LIN {X 0,Y 368.937,Z 294.527,A -85,B 0,C 180,E1 -12892.391,E2 -12892.391} C_VEL
LIN {X 0,Y 368.985,Z 294.519,A -85,B 0,C 180,E1 -12895.977,E2 -12895.977} C_VEL
LIN {X 0,Y 368.95,Z 294.527,A -85,B 0,C 180,E1 -12898.81,E2 -12898.81} C_VEL
LIN {X 0,Y 368.88,Z 294.532,A -85,B 0,C 180,E1 -12902.234,E2 -12902.234} C_VEL
LIN {X 0,Y 368.907,Z 294.534,A -85,B 0,C 180,E1 -12904.998,E2 -12904.998} C_VEL
LIN {X 0,Y 368.889,Z 294.533,A -85,B 0,C 180,E1 -12908.637,E2 -12908.637} C_VEL
LIN {X 0,Y 368.962,Z 294.67,A -85,B 0,C 180,E1 -12910.272,E2 -12910.272} C_VEL
LIN {X 0,Y 369.512,Z 297.416,A -85,B 0,C 180,E1 -12911.001,E2 -12911.001} C_VEL
LIN {X 0,Y 374.72,Z 313.747,A -85,B 0,C 180,E1 -12911.64,E2 -12911.64} C_VEL
LIN {X 0,Y 375.92,Z 320.785,A -85,B 0,C 180,E1 -12911.859,E2 -12911.859} C_VEL
LIN {X 0,Y 375.904,Z 322.653,A -85,B 0,C 180,E1 -12911.902,E2 -12911.902} C_VEL
LIN {X 0,Y 375.086,Z 328.475,A -85,B 0,C 180,E1 -12911.998,E2 -12911.998} C_VEL
LIN {X 0,Y 369.16,Z 347.372,A -85,B 0,C 180,E1 -12912.166,E2 -12912.166} C_VEL
LIN {X 0,Y 368.425,Z 353.191,A -85,B 0,C 180,E1 -12912.271,E2 -12912.271} C_VEL
LIN {X 0,Y 367.241,Z 406.595,A -85,B 0,C 180,E1 -12913.49,E2 -12913.49} C_VEL
LIN {X 0,Y 366.848,Z 418.98,A -85,B 0,C 180,E1 -12913.978,E2 -12913.978} C_VEL
LIN {X 0,Y 366.221,Z 431.276,A -85,B 0,C 180,E1 -12914.664,E2 -12914.664} C_VEL
LIN {X 0,Y 365.574,Z 442.837,A -85,B 0,C 180,E1 -12915.53,E2 -12915.53} C_VEL
LIN {X 0,Y 364.747,Z 453.885,A -85,B 0,C 180,E1 -12916.579,E2 -12916.579} C_VEL
LIN {X 0,Y 363.922,Z 464.624,A -85,B 0,C 180,E1 -12917.85,E2 -12917.85} C_VEL
LIN {X 0,Y 363.098,Z 474.262,A -85,B 0,C 180,E1 -12919.27,E2 -12919.27} C_VEL
LIN {X 0,Y 362.367,Z 483.022,A -85,B 0,C 180,E1 -12920.867,E2 -12920.867} C_VEL
LIN {X 0,Y 361.726,Z 490.562,A -85,B 0,C 180,E1 -12922.57,E2 -12922.57} C_VEL
LIN {X 0,Y 361.27,Z 496.591,A -85,B 0,C 180,E1 -12924.296,E2 -12924.296} C_VEL
LIN {X 0,Y 360.869,Z 501.916,A -85,B 0,C 180,E1 -12926.288,E2 -12926.288} C_VEL
LIN {X 0,Y 360.532,Z 505.675,A -85,B 0,C 180,E1 -12928.243,E2 -12928.243} C_VEL
LIN {X 0,Y 360.404,Z 507.362,A -85,B 0,C 180,E1 -12929.536,E2 -12929.536} C_VEL
LIN {X 0,Y 360.357,Z 508.805,A -85,B 0,C 180,E1 -12931.343,E2 -12931.343} C_VEL
LIN {X 0,Y 360.365,Z 509.152,A -85,B 0,C 180,E1 -12933.35,E2 -12933.35} C_VEL
LIN {X 0,Y 360.486,Z 508.683,A -85,B 0,C 180,E1 -12934.602,E2 -12934.602} C_VEL
LIN {X 0,Y 360.749,Z 507.241,A -85,B 0,C 180,E1 -12936.279,E2 -12936.279} C_VEL
LIN {X 0,Y 361.198,Z 504.193,A -85,B 0,C 180,E1 -12938.304,E2 -12938.304} C_VEL
LIN {X 0,Y 361.664,Z 500.21,A -85,B 0,C 180,E1 -12940.12,E2 -12940.12} C_VEL
LIN {X 0,Y 362.37,Z 494.924,A -85,B 0,C 180,E1 -12941.923,E2 -12941.923} C_VEL
LIN {X 0,Y 363.289,Z 488.133,A -85,B 0,C 180,E1 -12943.71,E2 -12943.71} C_VEL
LIN {X 0,Y 364.388,Z 479.592,A -85,B 0,C 180,E1 -12945.48,E2 -12945.48} C_VEL
LIN {X 0,Y 365.473,Z 470.795,A -85,B 0,C 180,E1 -12946.942,E2 -12946.942} C_VEL
LIN {X 0,Y 366.712,Z 460.323,A -85,B 0,C 180,E1 -12948.331,E2 -12948.331} C_VEL
LIN {X 0,Y 367.803,Z 449.016,A -85,B 0,C 180,E1 -12949.542,E2 -12949.542} C_VEL
LIN {X 0,Y 368.872,Z 436.91,A -85,B 0,C 180,E1 -12950.542,E2 -12950.542} C_VEL
LIN {X 0,Y 369.659,Z 424.92,A -85,B 0,C 180,E1 -12951.302,E2 -12951.302} C_VEL
LIN {X 0,Y 370.291,Z 412.735,A -85,B 0,C 180,E1 -12951.86,E2 -12951.86} C_VEL
LIN {X 0,Y 370.758,Z 397.567,A -85,B 0,C 180,E1 -12952.291,E2 -12952.291} C_VEL
LIN {X 0,Y 373.067,Z 321.948,A -85,B 0,C 180,E1 -12954.082,E2 -12954.082} C_VEL
LIN {X 0,Y 367.77,Z 308.846,A -85,B 0,C 180,E1 -12954.896,E2 -12954.896} C_VEL
LIN {X 0,Y 362.98,Z 299.287,A -85,B 0,C 180,E1 -12955.628,E2 -12955.628} C_VEL
LIN {X 0,Y 362.025,Z 295.396,A -85,B 0,C 180,E1 -12956.592,E2 -12956.592} C_VEL
LIN {X 0,Y 362.232,Z 295.369,A -85,B 0,C 180,E1 -12957.777,E2 -12957.777} C_VEL
LIN {X 0,Y 362.377,Z 295.346,A -85,B 0,C 180,E1 -12960.001,E2 -12960.001} C_VEL
LIN {X 0,Y 362.232,Z 295.365,A -85,B 0,C 180,E1 -12962.224,E2 -12962.224} C_VEL
LIN {X 0,Y 362.112,Z 295.379,A -85,B 0,C 180,E1 -12966.688,E2 -12966.688} C_VEL
LIN {X 0,Y 361.986,Z 295.393,A -85,B 0,C 180,E1 -12970.064,E2 -12970.064} C_VEL
LIN {X 0,Y 361.953,Z 295.398,A -85,B 0,C 180,E1 -12973.9,E2 -12973.9} C_VEL
LIN {X 0,Y 361.883,Z 295.406,A -85,B 0,C 180,E1 -12976.937,E2 -12976.937} C_VEL
LIN {X 0,Y 361.832,Z 295.407,A -85,B 0,C 180,E1 -12980.465,E2 -12980.465} C_VEL
LIN {X 0,Y 361.854,Z 295.409,A -85,B 0,C 180,E1 -12984.116,E2 -12984.116} C_VEL
LIN {X 0,Y 361.901,Z 295.401,A -85,B 0,C 180,E1 -12986.724,E2 -12986.724} C_VEL
LIN {X 0,Y 361.815,Z 295.415,A -85,B 0,C 180,E1 -12990.334,E2 -12990.334} C_VEL
LIN {X 0,Y 361.82,Z 295.41,A -85,B 0,C 180,E1 -12994.285,E2 -12994.285} C_VEL
LIN {X 0,Y 361.833,Z 295.41,A -85,B 0,C 180,E1 -12997.227,E2 -12997.227} C_VEL
LIN {X 0,Y 361.841,Z 295.412,A -85,B 0,C 180,E1 -13000.766,E2 -13000.766} C_VEL
LIN {X 0,Y 361.79,Z 295.416,A -85,B 0,C 180,E1 -13004.373,E2 -13004.373} C_VEL
LIN {X 0,Y 361.812,Z 295.419,A -85,B 0,C 180,E1 -13007.573,E2 -13007.573} C_VEL
LIN {X 0,Y 361.845,Z 295.412,A -85,B 0,C 180,E1 -13010.979,E2 -13010.979} C_VEL
LIN {X 0,Y 361.857,Z 295.415,A -85,B 0,C 180,E1 -13014.66,E2 -13014.66} C_VEL
LIN {X 0,Y 361.893,Z 295.418,A -85,B 0,C 180,E1 -13018.3,E2 -13018.3} C_VEL
LIN {X 0,Y 364.588,Z 305.964,A -85,B 0,C 180,E1 -13020.915,E2 -13020.915} C_VEL
LIN {X 0,Y 366.627,Z 315.872,A -85,B 0,C 180,E1 -13023.23,E2 -13023.23} C_VEL
LIN {X 0,Y 366.76,Z 318.771,A -85,B 0,C 180,E1 -13023.854,E2 -13023.854} C_VEL
LIN {X 0,Y 365.434,Z 332.937,A -85,B 0,C 180,E1 -13026.691,E2 -13026.691} C_VEL
LIN {X 0,Y 369.47,Z 354.155,A -85,B 0,C 180,E1 -13027.61,E2 -13027.61} C_VEL
LIN {X 0,Y 371.571,Z 370.409,A -85,B 0,C 180,E1 -13028.205,E2 -13028.205} C_VEL
LIN {X 0,Y 371.845,Z 375.745,A -85,B 0,C 180,E1 -13028.366,E2 -13028.366} C_VEL
LIN {X 0,Y 369.813,Z 444.426,A -85,B 0,C 180,E1 -13030.001,E2 -13030.001} C_VEL
LIN {X 0,Y 368.911,Z 458.053,A -85,B 0,C 180,E1 -13030.529,E2 -13030.529} C_VEL
LIN {X 0,Y 367.912,Z 470.015,A -85,B 0,C 180,E1 -13031.199,E2 -13031.199} C_VEL
LIN {X 0,Y 366.675,Z 482.615,A -85,B 0,C 180,E1 -13032.145,E2 -13032.145} C_VEL
LIN {X 0,Y 365.448,Z 493.967,A -85,B 0,C 180,E1 -13033.237,E2 -13033.237} C_VEL
LIN {X 0,Y 364.248,Z 504.34,A -85,B 0,C 180,E1 -13034.483,E2 -13034.483} C_VEL
LIN {X 0,Y 363.079,Z 514.461,A -85,B 0,C 180,E1 -13036.001,E2 -13036.001} C_VEL
LIN {X 0,Y 362.119,Z 523.48,A -85,B 0,C 180,E1 -13037.676,E2 -13037.676} C_VEL
LIN {X 0,Y 361.285,Z 530.704,A -85,B 0,C 180,E1 -13039.353,E2 -13039.353} C_VEL
LIN {X 0,Y 360.817,Z 536.522,A -85,B 0,C 180,E1 -13041.038,E2 -13041.038} C_VEL
LIN {X 0,Y 360.565,Z 541.13,A -85,B 0,C 180,E1 -13042.724,E2 -13042.724} C_VEL
LIN {X 0,Y 360.397,Z 544.627,A -85,B 0,C 180,E1 -13044.407,E2 -13044.407} C_VEL
LIN {X 0,Y 360.407,Z 546.388,A -85,B 0,C 180,E1 -13045.529,E2 -13045.529} C_VEL
LIN {X 0,Y 360.364,Z 547.727,A -85,B 0,C 180,E1 -13046.648,E2 -13046.648} C_VEL
LIN {X 0,Y 360.43,Z 548.607,A -85,B 0,C 180,E1 -13047.767,E2 -13047.767} C_VEL
LIN {X 0,Y 360.52,Z 549.064,A -85,B 0,C 180,E1 -13048.885,E2 -13048.885} C_VEL
LIN {X 0,Y 360.523,Z 549.11,A -85,B 0,C 180,E1 -13050.002,E2 -13050.002} C_VEL
LIN {X 0,Y 360.533,Z 548.742,A -85,B 0,C 180,E1 -13051.119,E2 -13051.119} C_VEL
LIN {X 0,Y 360.503,Z 547.904,A -85,B 0,C 180,E1 -13052.236,E2 -13052.236} C_VEL
LIN {X 0,Y 360.398,Z 546.633,A -85,B 0,C 180,E1 -13053.355,E2 -13053.355} C_VEL
LIN {X 0,Y 360.479,Z 543.903,A -85,B 0,C 180,E1 -13055.034,E2 -13055.034} C_VEL
LIN {X 0,Y 360.57,Z 540.082,A -85,B 0,C 180,E1 -13056.717,E2 -13056.717} C_VEL
LIN {X 0,Y 360.697,Z 535.07,A -85,B 0,C 180,E1 -13058.404,E2 -13058.404} C_VEL
LIN {X 0,Y 361.053,Z 528.729,A -85,B 0,C 180,E1 -13060.09,E2 -13060.09} C_VEL
LIN {X 0,Y 361.659,Z 520.778,A -85,B 0,C 180,E1 -13061.774,E2 -13061.774} C_VEL
LIN {X 0,Y 362.295,Z 512.626,A -85,B 0,C 180,E1 -13063.176,E2 -13063.176} C_VEL
LIN {X 0,Y 363.086,Z 502.676,A -85,B 0,C 180,E1 -13064.574,E2 -13064.574} C_VEL
LIN {X 0,Y 364.013,Z 491.591,A -85,B 0,C 180,E1 -13065.826,E2 -13065.826} C_VEL
LIN {X 0,Y 365.001,Z 479.007,A -85,B 0,C 180,E1 -13066.932,E2 -13066.932} C_VEL
LIN {X 0,Y 365.887,Z 466.723,A -85,B 0,C 180,E1 -13067.754,E2 -13067.754} C_VEL
LIN {X 0,Y 366.652,Z 453.074,A -85,B 0,C 180,E1 -13068.401,E2 -13068.401} C_VEL
LIN {X 0,Y 367.187,Z 439.632,A -85,B 0,C 180,E1 -13068.807,E2 -13068.807} C_VEL
LIN {X 0,Y 368.409,Z 371.766,A -85,B 0,C 180,E1 -13070.329,E2 -13070.329} C_VEL
LIN {X 0,Y 363.954,Z 336.994,A -85,B 0,C 180,E1 -13071.386,E2 -13071.386} C_VEL
LIN {X 0,Y 365.627,Z 318.277,A -85,B 0,C 180,E1 -13075.387,E2 -13075.387} C_VEL
LIN {X 0,Y 365.717,Z 314.433,A -85,B 0,C 180,E1 -13076.23,E2 -13076.23} C_VEL
LIN {X 0,Y 363.066,Z 300.891,A -85,B 0,C 180,E1 -13079.414,E2 -13079.414} C_VEL
LIN {X 0,Y 361.884,Z 295.409,A -85,B 0,C 180,E1 -13080.783,E2 -13080.783} C_VEL
LIN {X 0,Y 361.846,Z 295.412,A -85,B 0,C 180,E1 -13084.279,E2 -13084.279} C_VEL
LIN {X 0,Y 361.851,Z 295.41,A -85,B 0,C 180,E1 -13087.219,E2 -13087.219} C_VEL
LIN {X 0,Y 361.803,Z 295.42,A -85,B 0,C 180,E1 -13090.749,E2 -13090.749} C_VEL
LIN {X 0,Y 361.8,Z 295.416,A -85,B 0,C 180,E1 -13094.368,E2 -13094.368} C_VEL
LIN {X 0,Y 361.81,Z 295.414,A -85,B 0,C 180,E1 -13097.569,E2 -13097.569} C_VEL
LIN {X 0,Y 361.827,Z 295.412,A -85,B 0,C 180,E1 -13101.57,E2 -13101.57} C_VEL
LIN {X 0,Y 361.854,Z 295.411,A -85,B 0,C 180,E1 -13104.655,E2 -13104.655} C_VEL
LIN {X 0,Y 361.829,Z 295.416,A -85,B 0,C 180,E1 -13107.053,E2 -13107.053} C_VEL
LIN {X 0,Y 361.849,Z 295.414,A -85,B 0,C 180,E1 -13110.95,E2 -13110.95} C_VEL
LIN {X 0,Y 361.863,Z 295.409,A -85,B 0,C 180,E1 -13114.705,E2 -13114.705} C_VEL
LIN {X 0,Y 361.832,Z 295.411,A -85,B 0,C 180,E1 -13118.343,E2 -13118.343} C_VEL
LIN {X 0,Y 361.897,Z 295.403,A -85,B 0,C 180,E1 -13122.084,E2 -13122.084} C_VEL
LIN {X 0,Y 361.937,Z 295.402,A -85,B 0,C 180,E1 -13125.378,E2 -13125.378} C_VEL
LIN {X 0,Y 361.945,Z 295.398,A -85,B 0,C 180,E1 -13128.803,E2 -13128.803} C_VEL
LIN {X 0,Y 362.09,Z 295.379,A -85,B 0,C 180,E1 -13132.191,E2 -13132.191} C_VEL
LIN {X 0,Y 362.083,Z 295.38,A -85,B 0,C 180,E1 -13134.43,E2 -13134.43} C_VEL
LIN {X 0,Y 362.249,Z 295.362,A -85,B 0,C 180,E1 -13137.776,E2 -13137.776} C_VEL
LIN {X 0,Y 362.356,Z 295.347,A -85,B 0,C 180,E1 -13139.999,E2 -13139.999} C_VEL
LIN {X 0,Y 362.249,Z 295.36,A -85,B 0,C 180,E1 -13142.223,E2 -13142.223} C_VEL
LIN {X 0,Y 362.129,Z 295.374,A -85,B 0,C 180,E1 -13146.686,E2 -13146.686} C_VEL
LIN {X 0,Y 362.006,Z 295.391,A -85,B 0,C 180,E1 -13150.062,E2 -13150.062} C_VEL
LIN {X 0,Y 361.973,Z 295.397,A -85,B 0,C 180,E1 -13153.898,E2 -13153.898} C_VEL
LIN {X 0,Y 361.901,Z 295.403,A -85,B 0,C 180,E1 -13156.935,E2 -13156.935} C_VEL
LIN {X 0,Y 361.851,Z 295.409,A -85,B 0,C 180,E1 -13160.462,E2 -13160.462} C_VEL
LIN {X 0,Y 361.872,Z 295.409,A -85,B 0,C 180,E1 -13164.114,E2 -13164.114} C_VEL
LIN {X 0,Y 361.92,Z 295.4,A -85,B 0,C 180,E1 -13166.722,E2 -13166.722} C_VEL
LIN {X 0,Y 361.855,Z 295.41,A -85,B 0,C 180,E1 -13170.329,E2 -13170.329} C_VEL
LIN {X 0,Y 361.835,Z 295.414,A -85,B 0,C 180,E1 -13174.282,E2 -13174.282} C_VEL
LIN {X 0,Y 361.847,Z 295.41,A -85,B 0,C 180,E1 -13177.224,E2 -13177.224} C_VEL
LIN {X 0,Y 361.853,Z 295.409,A -85,B 0,C 180,E1 -13180.762,E2 -13180.762} C_VEL
LIN {X 0,Y 361.829,Z 295.415,A -85,B 0,C 180,E1 -13184.366,E2 -13184.366} C_VEL
LIN {X 0,Y 361.871,Z 295.408,A -85,B 0,C 180,E1 -13187.561,E2 -13187.561} C_VEL
LIN {X 0,Y 361.863,Z 295.408,A -85,B 0,C 180,E1 -13190.974,E2 -13190.974} C_VEL
LIN {X 0,Y 361.865,Z 295.409,A -85,B 0,C 180,E1 -13194.656,E2 -13194.656} C_VEL
LIN {X 0,Y 361.83,Z 295.416,A -85,B 0,C 180,E1 -13198.371,E2 -13198.371} C_VEL
LIN {X 0,Y 361.902,Z 295.406,A -85,B 0,C 180,E1 -13202.221,E2 -13202.221} C_VEL
LIN {X 0,Y 361.923,Z 295.402,A -85,B 0,C 180,E1 -13204.71,E2 -13204.71} C_VEL
LIN {X 0,Y 361.888,Z 295.408,A -85,B 0,C 180,E1 -13208.347,E2 -13208.347} C_VEL
LIN {X 0,Y 361.964,Z 295.398,A -85,B 0,C 180,E1 -13212.061,E2 -13212.061} C_VEL
LIN {X 0,Y 361.995,Z 295.394,A -85,B 0,C 180,E1 -13216.101,E2 -13216.101} C_VEL
LIN {X 0,Y 362.029,Z 295.388,A -85,B 0,C 180,E1 -13219.937,E2 -13219.937} C_VEL
LIN {X 0,Y 362.149,Z 295.374,A -85,B 0,C 180,E1 -13222.192,E2 -13222.192} C_VEL
LIN {X 0,Y 362.116,Z 295.379,A -85,B 0,C 180,E1 -13224.43,E2 -13224.43} C_VEL
LIN {X 0,Y 362.28,Z 295.355,A -85,B 0,C 180,E1 -13227.775,E2 -13227.775} C_VEL
LIN {X 0,Y 362.425,Z 295.338,A -85,B 0,C 180,E1 -13229.998,E2 -13229.998} C_VEL
LIN {X 0,Y 362.28,Z 295.357,A -85,B 0,C 180,E1 -13232.222,E2 -13232.222} C_VEL
LIN {X 0,Y 362.165,Z 295.374,A -85,B 0,C 180,E1 -13236.684,E2 -13236.684} C_VEL
LIN {X 0,Y 362.069,Z 295.386,A -85,B 0,C 180,E1 -13238.931,E2 -13238.931} C_VEL
LIN {X 0,Y 361.959,Z 295.397,A -85,B 0,C 180,E1 -13242.329,E2 -13242.329} C_VEL
LIN {X 0,Y 361.954,Z 295.399,A -85,B 0,C 180,E1 -13244.617,E2 -13244.617} C_VEL
LIN {X 0,Y 361.951,Z 295.396,A -85,B 0,C 180,E1 -13248.096,E2 -13248.096} C_VEL
LIN {X 0,Y 361.902,Z 295.402,A -85,B 0,C 180,E1 -13251.648,E2 -13251.648} C_VEL
LIN {X 0,Y 361.914,Z 295.403,A -85,B 0,C 180,E1 -13255.286,E2 -13255.286} C_VEL
LIN {X 0,Y 361.906,Z 295.401,A -85,B 0,C 180,E1 -13257.774,E2 -13257.774} C_VEL
LIN {X 0,Y 361.828,Z 295.415,A -85,B 0,C 180,E1 -13261.282,E2 -13261.282} C_VEL
LIN {X 0,Y 361.833,Z 295.41,A -85,B 0,C 180,E1 -13264.277,E2 -13264.277} C_VEL
LIN {X 0,Y 361.848,Z 295.414,A -85,B 0,C 180,E1 -13267.221,E2 -13267.221} C_VEL
LIN {X 0,Y 361.916,Z 295.43,A -85,B 0,C 180,E1 -13270.017,E2 -13270.017} C_VEL
LIN {X 0,Y 362.382,Z 297.887,A -85,B 0,C 180,E1 -13270.663,E2 -13270.663} C_VEL
LIN {X 0,Y 368.104,Z 315.692,A -85,B 0,C 180,E1 -13271.374,E2 -13271.374} C_VEL
LIN {X 0,Y 369.116,Z 321.233,A -85,B 0,C 180,E1 -13271.554,E2 -13271.554} C_VEL
LIN {X 0,Y 368.425,Z 353.191,A -85,B 0,C 180,E1 -13272.271,E2 -13272.271} C_VEL
LIN {X 0,Y 367.673,Z 359.015,A -85,B 0,C 180,E1 -13272.374,E2 -13272.374} C_VEL
LIN {X 0,Y 361.662,Z 377.908,A -85,B 0,C 180,E1 -13272.548,E2 -13272.548} C_VEL
LIN {X 0,Y 360.879,Z 383.734,A -85,B 0,C 180,E1 -13272.652,E2 -13272.652} C_VEL
LIN {X 0,Y 360.342,Z 407.807,A -85,B 0,C 180,E1 -13273.244,E2 -13273.244} C_VEL
LIN {X 0,Y 359.954,Z 420.001,A -85,B 0,C 180,E1 -13273.747,E2 -13273.747} C_VEL
LIN {X 0,Y 359.306,Z 432.235,A -85,B 0,C 180,E1 -13274.454,E2 -13274.454} C_VEL
LIN {X 0,Y 358.622,Z 443.582,A -85,B 0,C 180,E1 -13275.329,E2 -13275.329} C_VEL
LIN {X 0,Y 357.785,Z 454.352,A -85,B 0,C 180,E1 -13276.374,E2 -13276.374} C_VEL
LIN {X 0,Y 356.973,Z 464.554,A -85,B 0,C 180,E1 -13277.601,E2 -13277.601} C_VEL
LIN {X 0,Y 356.132,Z 474.289,A -85,B 0,C 180,E1 -13279.045,E2 -13279.045} C_VEL
LIN {X 0,Y 355.332,Z 483.423,A -85,B 0,C 180,E1 -13280.735,E2 -13280.735} C_VEL
LIN {X 0,Y 354.687,Z 490.753,A -85,B 0,C 180,E1 -13282.417,E2 -13282.417} C_VEL
LIN {X 0,Y 354.243,Z 496.343,A -85,B 0,C 180,E1 -13284.014,E2 -13284.014} C_VEL
LIN {X 0,Y 353.898,Z 500.604,A -85,B 0,C 180,E1 -13285.531,E2 -13285.531} C_VEL
LIN {X 0,Y 353.769,Z 502.956,A -85,B 0,C 180,E1 -13286.539,E2 -13286.539} C_VEL
LIN {X 0,Y 353.567,Z 504.904,A -85,B 0,C 180,E1 -13287.542,E2 -13287.542} C_VEL
LIN {X 0,Y 353.376,Z 506.929,A -85,B 0,C 180,E1 -13288.863,E2 -13288.863} C_VEL
LIN {X 0,Y 353.28,Z 509.047,A -85,B 0,C 180,E1 -13291.068,E2 -13291.068} C_VEL
LIN {X 0,Y 353.275,Z 509.616,A -85,B 0,C 180,E1 -13292.771,E2 -13292.771} C_VEL
LIN {X 0,Y 353.357,Z 509.404,A -85,B 0,C 180,E1 -13294.052,E2 -13294.052} C_VEL
LIN {X 0,Y 353.625,Z 508.047,A -85,B 0,C 180,E1 -13296.076,E2 -13296.076} C_VEL
LIN {X 0,Y 354.027,Z 505.768,A -85,B 0,C 180,E1 -13297.842,E2 -13297.842} C_VEL
LIN {X 0,Y 354.491,Z 502.228,A -85,B 0,C 180,E1 -13299.7,E2 -13299.7} C_VEL
LIN {X 0,Y 355.227,Z 496.869,A -85,B 0,C 180,E1 -13301.719,E2 -13301.719} C_VEL
LIN {X 0,Y 356.237,Z 489.977,A -85,B 0,C 180,E1 -13303.673,E2 -13303.673} C_VEL
LIN {X 0,Y 357.363,Z 481.801,A -85,B 0,C 180,E1 -13305.479,E2 -13305.479} C_VEL
LIN {X 0,Y 358.469,Z 473.4,A -85,B 0,C 180,E1 -13306.97,E2 -13306.97} C_VEL
LIN {X 0,Y 359.681,Z 463.925,A -85,B 0,C 180,E1 -13308.339,E2 -13308.339} C_VEL
LIN {X 0,Y 360.948,Z 452.806,A -85,B 0,C 180,E1 -13309.625,E2 -13309.625} C_VEL
LIN {X 0,Y 361.948,Z 441.756,A -85,B 0,C 180,E1 -13310.642,E2 -13310.642} C_VEL
LIN {X 0,Y 362.973,Z 429.197,A -85,B 0,C 180,E1 -13311.532,E2 -13311.532} C_VEL
LIN {X 0,Y 363.688,Z 416.105,A -85,B 0,C 180,E1 -13312.201,E2 -13312.201} C_VEL
LIN {X 0,Y 364.188,Z 403.673,A -85,B 0,C 180,E1 -13312.621,E2 -13312.621} C_VEL
LIN {X 0,Y 366.868,Z 323.745,A -85,B 0,C 180,E1 -13314.561,E2 -13314.561} C_VEL
LIN {X 0,Y 361.403,Z 310.693,A -85,B 0,C 180,E1 -13315.422,E2 -13315.422} C_VEL
LIN {X 0,Y 355.957,Z 299.947,A -85,B 0,C 180,E1 -13316.286,E2 -13316.286} C_VEL
LIN {X 0,Y 355.09,Z 296.259,A -85,B 0,C 180,E1 -13317.235,E2 -13317.235} C_VEL
LIN {X 0,Y 355.326,Z 296.224,A -85,B 0,C 180,E1 -13320.001,E2 -13320.001} C_VEL
LIN {X 0,Y 355.196,Z 296.242,A -85,B 0,C 180,E1 -13322.268,E2 -13322.268} C_VEL
LIN {X 0,Y 355.076,Z 296.256,A -85,B 0,C 180,E1 -13326.821,E2 -13326.821} C_VEL
LIN {X 0,Y 354.933,Z 296.271,A -85,B 0,C 180,E1 -13330.266,E2 -13330.266} C_VEL
LIN {X 0,Y 354.898,Z 296.277,A -85,B 0,C 180,E1 -13334.02,E2 -13334.02} C_VEL
LIN {X 0,Y 354.846,Z 296.279,A -85,B 0,C 180,E1 -13338.094,E2 -13338.094} C_VEL
LIN {X 0,Y 354.775,Z 296.29,A -85,B 0,C 180,E1 -13342.11,E2 -13342.11} C_VEL
LIN {X 0,Y 354.858,Z 296.276,A -85,B 0,C 180,E1 -13345.831,E2 -13345.831} C_VEL
LIN {X 0,Y 354.766,Z 296.294,A -85,B 0,C 180,E1 -13349.687,E2 -13349.687} C_VEL
LIN {X 0,Y 354.782,Z 296.289,A -85,B 0,C 180,E1 -13353.688,E2 -13353.688} C_VEL
LIN {X 0,Y 354.766,Z 296.293,A -85,B 0,C 180,E1 -13356.464,E2 -13356.464} C_VEL
LIN {X 0,Y 354.796,Z 296.287,A -85,B 0,C 180,E1 -13359.428,E2 -13359.428} C_VEL
LIN {X 0,Y 354.764,Z 296.291,A -85,B 0,C 180,E1 -13362.872,E2 -13362.872} C_VEL
LIN {X 0,Y 354.742,Z 296.296,A -85,B 0,C 180,E1 -13366.108,E2 -13366.108} C_VEL
LIN {X 0,Y 354.765,Z 296.294,A -85,B 0,C 180,E1 -13369.183,E2 -13369.183} C_VEL
LIN {X 0,Y 354.787,Z 296.291,A -85,B 0,C 180,E1 -13372.408,E2 -13372.408} C_VEL
LIN {X 0,Y 354.795,Z 296.294,A -85,B 0,C 180,E1 -13374.945,E2 -13374.945} C_VEL
LIN {X 0,Y 354.837,Z 296.474,A -85,B 0,C 180,E1 -13377.742,E2 -13377.742} C_VEL
LIN {X 0,Y 357.778,Z 307.54,A -85,B 0,C 180,E1 -13380.593,E2 -13380.593} C_VEL
LIN {X 0,Y 359.847,Z 317.585,A -85,B 0,C 180,E1 -13382.999,E2 -13382.999} C_VEL
LIN {X 0,Y 359.951,Z 321.077,A -85,B 0,C 180,E1 -13383.761,E2 -13383.761} C_VEL
LIN {X 0,Y 358.818,Z 332.325,A -85,B 0,C 180,E1 -13386.061,E2 -13386.061} C_VEL
LIN {X 0,Y 363.163,Z 354.917,A -85,B 0,C 180,E1 -13387.101,E2 -13387.101} C_VEL
LIN {X 0,Y 365.307,Z 372.289,A -85,B 0,C 180,E1 -13387.764,E2 -13387.764} C_VEL
LIN {X 0,Y 365.446,Z 377.924,A -85,B 0,C 180,E1 -13387.927,E2 -13387.927} C_VEL
LIN {X 0,Y 363.404,Z 443.639,A -85,B 0,C 180,E1 -13389.522,E2 -13389.522} C_VEL
LIN {X 0,Y 362.478,Z 457.338,A -85,B 0,C 180,E1 -13390.059,E2 -13390.059} C_VEL
LIN {X 0,Y 361.336,Z 469.887,A -85,B 0,C 180,E1 -13390.769,E2 -13390.769} C_VEL
LIN {X 0,Y 359.962,Z 483.144,A -85,B 0,C 180,E1 -13391.801,E2 -13391.801} C_VEL
LIN {X 0,Y 358.664,Z 494.275,A -85,B 0,C 180,E1 -13392.911,E2 -13392.911} C_VEL
LIN {X 0,Y 357.391,Z 504.603,A -85,B 0,C 180,E1 -13394.203,E2 -13394.203} C_VEL
LIN {X 0,Y 356.168,Z 514.479,A -85,B 0,C 180,E1 -13395.724,E2 -13395.724} C_VEL
LIN {X 0,Y 355.346,Z 522.034,A -85,B 0,C 180,E1 -13397.147,E2 -13397.147} C_VEL
LIN {X 0,Y 354.358,Z 529.502,A -85,B 0,C 180,E1 -13398.853,E2 -13398.853} C_VEL
LIN {X 0,Y 353.908,Z 534.566,A -85,B 0,C 180,E1 -13400.285,E2 -13400.285} C_VEL
LIN {X 0,Y 353.538,Z 539.511,A -85,B 0,C 180,E1 -13402.004,E2 -13402.004} C_VEL
LIN {X 0,Y 353.332,Z 543.851,A -85,B 0,C 180,E1 -13404.009,E2 -13404.009} C_VEL
LIN {X 0,Y 353.316,Z 546.071,A -85,B 0,C 180,E1 -13405.439,E2 -13405.439} C_VEL
LIN {X 0,Y 353.283,Z 547.382,A -85,B 0,C 180,E1 -13406.581,E2 -13406.581} C_VEL
LIN {X 0,Y 353.332,Z 548.229,A -85,B 0,C 180,E1 -13407.722,E2 -13407.722} C_VEL
LIN {X 0,Y 353.454,Z 548.67,A -85,B 0,C 180,E1 -13408.863,E2 -13408.863} C_VEL
LIN {X 0,Y 353.458,Z 548.695,A -85,B 0,C 180,E1 -13410.002,E2 -13410.002} C_VEL
LIN {X 0,Y 353.468,Z 548.29,A -85,B 0,C 180,E1 -13411.141,E2 -13411.141} C_VEL
LIN {X 0,Y 353.406,Z 547.418,A -85,B 0,C 180,E1 -13412.281,E2 -13412.281} C_VEL
LIN {X 0,Y 353.317,Z 546.125,A -85,B 0,C 180,E1 -13413.423,E2 -13413.423} C_VEL
LIN {X 0,Y 353.395,Z 543.341,A -85,B 0,C 180,E1 -13415.136,E2 -13415.136} C_VEL
LIN {X 0,Y 353.501,Z 539.463,A -85,B 0,C 180,E1 -13416.852,E2 -13416.852} C_VEL
LIN {X 0,Y 353.637,Z 534.384,A -85,B 0,C 180,E1 -13418.573,E2 -13418.573} C_VEL
LIN {X 0,Y 353.988,Z 527.966,A -85,B 0,C 180,E1 -13420.294,E2 -13420.294} C_VEL
LIN {X 0,Y 354.643,Z 519.896,A -85,B 0,C 180,E1 -13422.01,E2 -13422.01} C_VEL
LIN {X 0,Y 355.355,Z 511.648,A -85,B 0,C 180,E1 -13423.438,E2 -13423.438} C_VEL
LIN {X 0,Y 356.146,Z 501.57,A -85,B 0,C 180,E1 -13424.865,E2 -13424.865} C_VEL
LIN {X 0,Y 357.113,Z 490.252,A -85,B 0,C 180,E1 -13426.14,E2 -13426.14} C_VEL
LIN {X 0,Y 358.018,Z 479.216,A -85,B 0,C 180,E1 -13427.125,E2 -13427.125} C_VEL
LIN {X 0,Y 358.924,Z 467.128,A -85,B 0,C 180,E1 -13427.963,E2 -13427.963} C_VEL
LIN {X 0,Y 359.729,Z 453.895,A -85,B 0,C 180,E1 -13428.621,E2 -13428.621} C_VEL
LIN {X 0,Y 360.307,Z 439.85,A -85,B 0,C 180,E1 -13429.07,E2 -13429.07} C_VEL
LIN {X 0,Y 361.604,Z 372.698,A -85,B 0,C 180,E1 -13430.611,E2 -13430.611} C_VEL
LIN {X 0,Y 357.007,Z 336.655,A -85,B 0,C 180,E1 -13431.736,E2 -13431.736} C_VEL
LIN {X 0,Y 358.655,Z 319.193,A -85,B 0,C 180,E1 -13435.537,E2 -13435.537} C_VEL
LIN {X 0,Y 358.844,Z 316.438,A -85,B 0,C 180,E1 -13436.145,E2 -13436.145} C_VEL
LIN {X 0,Y 356.436,Z 303.633,A -85,B 0,C 180,E1 -13439.208,E2 -13439.208} C_VEL
LIN {X 0,Y 354.808,Z 296.29,A -85,B 0,C 180,E1 -13441.051,E2 -13441.051} C_VEL
LIN {X 0,Y 354.803,Z 296.289,A -85,B 0,C 180,E1 -13445.058,E2 -13445.058} C_VEL
LIN {X 0,Y 354.786,Z 296.288,A -85,B 0,C 180,E1 -13447.883,E2 -13447.883} C_VEL
LIN {X 0,Y 354.759,Z 296.294,A -85,B 0,C 180,E1 -13451.165,E2 -13451.165} C_VEL
LIN {X 0,Y 354.747,Z 296.296,A -85,B 0,C 180,E1 -13454.503,E2 -13454.503} C_VEL
LIN {X 0,Y 354.77,Z 296.29,A -85,B 0,C 180,E1 -13457.658,E2 -13457.658} C_VEL
LIN {X 0,Y 354.774,Z 296.293,A -85,B 0,C 180,E1 -13460.66,E2 -13460.66} C_VEL
LIN {X 0,Y 354.803,Z 296.287,A -85,B 0,C 180,E1 -13464.3,E2 -13464.3} C_VEL
LIN {X 0,Y 354.763,Z 296.292,A -85,B 0,C 180,E1 -13467.664,E2 -13467.664} C_VEL
LIN {X 0,Y 354.792,Z 296.289,A -85,B 0,C 180,E1 -13471.613,E2 -13471.613} C_VEL
LIN {X 0,Y 354.816,Z 296.286,A -85,B 0,C 180,E1 -13475.655,E2 -13475.655} C_VEL
LIN {X 0,Y 354.8,Z 296.292,A -85,B 0,C 180,E1 -13479.111,E2 -13479.111} C_VEL
LIN {X 0,Y 354.857,Z 296.281,A -85,B 0,C 180,E1 -13482.717,E2 -13482.717} C_VEL
LIN {X 0,Y 354.927,Z 296.271,A -85,B 0,C 180,E1 -13486.254,E2 -13486.254} C_VEL
LIN {X 0,Y 354.933,Z 296.273,A -85,B 0,C 180,E1 -13489.734,E2 -13489.734} C_VEL
LIN {X 0,Y 355.096,Z 296.254,A -85,B 0,C 180,E1 -13493.179,E2 -13493.179} C_VEL
LIN {X 0,Y 355.213,Z 296.239,A -85,B 0,C 180,E1 -13497.732,E2 -13497.732} C_VEL
LIN {X 0,Y 355.307,Z 296.225,A -85,B 0,C 180,E1 -13499.999,E2 -13499.999} C_VEL
LIN {X 0,Y 355.212,Z 296.236,A -85,B 0,C 180,E1 -13502.267,E2 -13502.267} C_VEL
LIN {X 0,Y 355.094,Z 296.251,A -85,B 0,C 180,E1 -13506.819,E2 -13506.819} C_VEL
LIN {X 0,Y 354.954,Z 296.269,A -85,B 0,C 180,E1 -13510.264,E2 -13510.264} C_VEL
LIN {X 0,Y 354.918,Z 296.275,A -85,B 0,C 180,E1 -13514.018,E2 -13514.018} C_VEL
LIN {X 0,Y 354.853,Z 296.283,A -85,B 0,C 180,E1 -13517.282,E2 -13517.282} C_VEL
LIN {X 0,Y 354.795,Z 296.291,A -85,B 0,C 180,E1 -13521.418,E2 -13521.418} C_VEL
LIN {X 0,Y 354.839,Z 296.282,A -85,B 0,C 180,E1 -13524.577,E2 -13524.577} C_VEL
LIN {X 0,Y 354.863,Z 296.28,A -85,B 0,C 180,E1 -13527.097,E2 -13527.097} C_VEL
LIN {X 0,Y 354.834,Z 296.287,A -85,B 0,C 180,E1 -13529.68,E2 -13529.68} C_VEL
LIN {X 0,Y 354.789,Z 296.293,A -85,B 0,C 180,E1 -13533.703,E2 -13533.703} C_VEL
LIN {X 0,Y 354.78,Z 296.291,A -85,B 0,C 180,E1 -13536.461,E2 -13536.461} C_VEL
LIN {X 0,Y 354.809,Z 296.287,A -85,B 0,C 180,E1 -13539.425,E2 -13539.425} C_VEL
LIN {X 0,Y 354.777,Z 296.29,A -85,B 0,C 180,E1 -13542.869,E2 -13542.869} C_VEL
LIN {X 0,Y 354.825,Z 296.288,A -85,B 0,C 180,E1 -13546.116,E2 -13546.116} C_VEL
LIN {X 0,Y 354.845,Z 296.281,A -85,B 0,C 180,E1 -13549.19,E2 -13549.19} C_VEL
LIN {X 0,Y 354.803,Z 296.29,A -85,B 0,C 180,E1 -13552.403,E2 -13552.403} C_VEL
LIN {X 0,Y 354.803,Z 296.287,A -85,B 0,C 180,E1 -13554.942,E2 -13554.942} C_VEL
LIN {X 0,Y 354.786,Z 296.293,A -85,B 0,C 180,E1 -13558.406,E2 -13558.406} C_VEL
LIN {X 0,Y 354.84,Z 296.283,A -85,B 0,C 180,E1 -13561.619,E2 -13561.619} C_VEL
LIN {X 0,Y 354.893,Z 296.279,A -85,B 0,C 180,E1 -13564.173,E2 -13564.173} C_VEL
LIN {X 0,Y 354.83,Z 296.285,A -85,B 0,C 180,E1 -13567.894,E2 -13567.894} C_VEL
LIN {X 0,Y 354.92,Z 296.273,A -85,B 0,C 180,E1 -13571.891,E2 -13571.891} C_VEL
LIN {X 0,Y 354.94,Z 296.271,A -85,B 0,C 180,E1 -13575.981,E2 -13575.981} C_VEL
LIN {X 0,Y 354.976,Z 296.265,A -85,B 0,C 180,E1 -13579.735,E2 -13579.735} C_VEL
LIN {X 0,Y 355.112,Z 296.25,A -85,B 0,C 180,E1 -13582.036,E2 -13582.036} C_VEL
LIN {X 0,Y 355.09,Z 296.254,A -85,B 0,C 180,E1 -13584.319,E2 -13584.319} C_VEL
LIN {X 0,Y 355.243,Z 296.232,A -85,B 0,C 180,E1 -13587.731,E2 -13587.731} C_VEL
LIN {X 0,Y 355.395,Z 296.213,A -85,B 0,C 180,E1 -13589.998,E2 -13589.998} C_VEL
LIN {X 0,Y 355.243,Z 296.234,A -85,B 0,C 180,E1 -13592.266,E2 -13592.266} C_VEL
LIN {X 0,Y 355.131,Z 296.251,A -85,B 0,C 180,E1 -13596.817,E2 -13596.817} C_VEL
LIN {X 0,Y 355.01,Z 296.263,A -85,B 0,C 180,E1 -13599.11,E2 -13599.11} C_VEL
LIN {X 0,Y 354.919,Z 296.275,A -85,B 0,C 180,E1 -13602.578,E2 -13602.578} C_VEL
LIN {X 0,Y 354.881,Z 296.277,A -85,B 0,C 180,E1 -13606.093,E2 -13606.093} C_VEL
LIN {X 0,Y 354.9,Z 296.276,A -85,B 0,C 180,E1 -13608.468,E2 -13608.468} C_VEL
LIN {X 0,Y 354.838,Z 296.282,A -85,B 0,C 180,E1 -13612.101,E2 -13612.101} C_VEL
LIN {X 0,Y 354.885,Z 296.276,A -85,B 0,C 180,E1 -13615.824,E2 -13615.824} C_VEL
LIN {X 0,Y 354.837,Z 296.282,A -85,B 0,C 180,E1 -13619.675,E2 -13619.675} C_VEL
LIN {X 0,Y 354.786,Z 296.289,A -85,B 0,C 180,E1 -13623.698,E2 -13623.698} C_VEL
LIN {X 0,Y 354.778,Z 296.289,A -85,B 0,C 180,E1 -13626.455,E2 -13626.455} C_VEL
LIN {X 0,Y 354.891,Z 296.419,A -85,B 0,C 180,E1 -13629.816,E2 -13629.816} C_VEL
LIN {X 0,Y 355.217,Z 298.169,A -85,B 0,C 180,E1 -13630.294,E2 -13630.294} C_VEL
LIN {X 0,Y 361.639,Z 318.261,A -85,B 0,C 180,E1 -13631.121,E2 -13631.121} C_VEL
LIN {X 0,Y 362.327,Z 323.016,A -85,B 0,C 180,E1 -13631.27,E2 -13631.27} C_VEL
LIN {X 0,Y 360.879,Z 383.734,A -85,B 0,C 180,E1 -13632.652,E2 -13632.652} C_VEL
LIN {X 0,Y 360.085,Z 389.568,A -85,B 0,C 180,E1 -13632.752,E2 -13632.752} C_VEL
LIN {X 0,Y 353.964,Z 408.399,A -85,B 0,C 180,E1 -13632.992,E2 -13632.992} C_VEL
LIN {X 0,Y 353.239,Z 414.124,A -85,B 0,C 180,E1 -13633.19,E2 -13633.19} C_VEL
LIN {X 0,Y 352.728,Z 427.324,A -85,B 0,C 180,E1 -13633.862,E2 -13633.862} C_VEL
LIN {X 0,Y 351.959,Z 439.96,A -85,B 0,C 180,E1 -13634.756,E2 -13634.756} C_VEL
LIN {X 0,Y 351.04,Z 452.309,A -85,B 0,C 180,E1 -13635.894,E2 -13635.894} C_VEL
LIN {X 0,Y 350.085,Z 463.887,A -85,B 0,C 180,E1 -13637.271,E2 -13637.271} C_VEL
LIN {X 0,Y 349.188,Z 473.986,A -85,B 0,C 180,E1 -13638.766,E2 -13638.766} C_VEL
LIN {X 0,Y 348.44,Z 482.207,A -85,B 0,C 180,E1 -13640.271,E2 -13640.271} C_VEL
LIN {X 0,Y 347.699,Z 489.94,A -85,B 0,C 180,E1 -13642.017,E2 -13642.017} C_VEL
LIN {X 0,Y 347.215,Z 495.928,A -85,B 0,C 180,E1 -13643.698,E2 -13643.698} C_VEL
LIN {X 0,Y 346.841,Z 500.84,A -85,B 0,C 180,E1 -13645.434,E2 -13645.434} C_VEL
LIN {X 0,Y 346.498,Z 505.205,A -85,B 0,C 180,E1 -13647.487,E2 -13647.487} C_VEL
LIN {X 0,Y 346.216,Z 508.061,A -85,B 0,C 180,E1 -13649.504,E2 -13649.504} C_VEL
LIN {X 0,Y 346.205,Z 509.259,A -85,B 0,C 180,E1 -13650.844,E2 -13650.844} C_VEL
LIN {X 0,Y 346.167,Z 509.892,A -85,B 0,C 180,E1 -13652.164,E2 -13652.164} C_VEL
LIN {X 0,Y 346.209,Z 509.991,A -85,B 0,C 180,E1 -13653.475,E2 -13653.475} C_VEL
LIN {X 0,Y 346.365,Z 509.587,A -85,B 0,C 180,E1 -13654.78,E2 -13654.78} C_VEL
LIN {X 0,Y 346.543,Z 508.633,A -85,B 0,C 180,E1 -13656.072,E2 -13656.072} C_VEL
LIN {X 0,Y 346.826,Z 507.209,A -85,B 0,C 180,E1 -13657.356,E2 -13657.356} C_VEL
LIN {X 0,Y 347.337,Z 504.075,A -85,B 0,C 180,E1 -13659.263,E2 -13659.263} C_VEL
LIN {X 0,Y 347.946,Z 499.719,A -85,B 0,C 180,E1 -13661.146,E2 -13661.146} C_VEL
LIN {X 0,Y 348.827,Z 494.027,A -85,B 0,C 180,E1 -13663.015,E2 -13663.015} C_VEL
LIN {X 0,Y 349.94,Z 486.825,A -85,B 0,C 180,E1 -13664.866,E2 -13664.866} C_VEL
LIN {X 0,Y 351.023,Z 479.401,A -85,B 0,C 180,E1 -13666.394,E2 -13666.394} C_VEL
LIN {X 0,Y 352.365,Z 469.485,A -85,B 0,C 180,E1 -13668.035,E2 -13668.035} C_VEL
LIN {X 0,Y 353.769,Z 459.051,A -85,B 0,C 180,E1 -13669.412,E2 -13669.412} C_VEL
LIN {X 0,Y 354.957,Z 447.743,A -85,B 0,C 180,E1 -13670.599,E2 -13670.599} C_VEL
LIN {X 0,Y 356.007,Z 436.401,A -85,B 0,C 180,E1 -13671.538,E2 -13671.538} C_VEL
LIN {X 0,Y 356.853,Z 424.657,A -85,B 0,C 180,E1 -13672.29,E2 -13672.29} C_VEL
LIN {X 0,Y 357.533,Z 411.786,A -85,B 0,C 180,E1 -13672.873,E2 -13672.873} C_VEL
LIN {X 0,Y 358.23,Z 391.899,A -85,B 0,C 180,E1 -13673.417,E2 -13673.417} C_VEL
LIN {X 0,Y 360.532,Z 325.381,A -85,B 0,C 180,E1 -13675.083,E2 -13675.083} C_VEL
LIN {X 0,Y 355.519,Z 313.528,A -85,B 0,C 180,E1 -13675.909,E2 -13675.909} C_VEL
LIN {X 0,Y 348.906,Z 300.509,A -85,B 0,C 180,E1 -13677.006,E2 -13677.006} C_VEL
LIN {X 0,Y 348.137,Z 297.125,A -85,B 0,C 180,E1 -13677.904,E2 -13677.904} C_VEL
LIN {X 0,Y 348.276,Z 297.102,A -85,B 0,C 180,E1 -13680.001,E2 -13680.001} C_VEL
LIN {X 0,Y 348.159,Z 297.118,A -85,B 0,C 180,E1 -13682.314,E2 -13682.314} C_VEL
LIN {X 0,Y 348.042,Z 297.133,A -85,B 0,C 180,E1 -13686.959,E2 -13686.959} C_VEL
LIN {X 0,Y 347.885,Z 297.148,A -85,B 0,C 180,E1 -13690.476,E2 -13690.476} C_VEL
LIN {X 0,Y 347.856,Z 297.154,A -85,B 0,C 180,E1 -13694.152,E2 -13694.152} C_VEL
LIN {X 0,Y 347.786,Z 297.158,A -85,B 0,C 180,E1 -13698.261,E2 -13698.261} C_VEL
LIN {X 0,Y 347.726,Z 297.17,A -85,B 0,C 180,E1 -13701.629,E2 -13701.629} C_VEL
LIN {X 0,Y 347.772,Z 297.163,A -85,B 0,C 180,E1 -13705.112,E2 -13705.112} C_VEL
LIN {X 0,Y 347.764,Z 297.165,A -85,B 0,C 180,E1 -13707.698,E2 -13707.698} C_VEL
LIN {X 0,Y 347.706,Z 297.168,A -85,B 0,C 180,E1 -13711.704,E2 -13711.704} C_VEL
LIN {X 0,Y 347.712,Z 297.167,A -85,B 0,C 180,E1 -13714.468,E2 -13714.468} C_VEL
LIN {X 0,Y 347.745,Z 297.168,A -85,B 0,C 180,E1 -13717.993,E2 -13717.993} C_VEL
LIN {X 0,Y 347.732,Z 297.166,A -85,B 0,C 180,E1 -13721.834,E2 -13721.834} C_VEL
LIN {X 0,Y 347.679,Z 297.175,A -85,B 0,C 180,E1 -13725.032,E2 -13725.032} C_VEL
LIN {X 0,Y 347.728,Z 297.17,A -85,B 0,C 180,E1 -13728.402,E2 -13728.402} C_VEL
LIN {X 0,Y 347.753,Z 297.166,A -85,B 0,C 180,E1 -13732.017,E2 -13732.017} C_VEL
LIN {X 0,Y 347.728,Z 297.178,A -85,B 0,C 180,E1 -13735.541,E2 -13735.541} C_VEL
LIN {X 0,Y 347.761,Z 297.32,A -85,B 0,C 180,E1 -13737.082,E2 -13737.082} C_VEL
LIN {X 0,Y 350.7,Z 307.97,A -85,B 0,C 180,E1 -13739.939,E2 -13739.939} C_VEL
LIN {X 0,Y 352.817,Z 317.986,A -85,B 0,C 180,E1 -13742.436,E2 -13742.436} C_VEL
LIN {X 0,Y 353.297,Z 321.926,A -85,B 0,C 180,E1 -13743.354,E2 -13743.354} C_VEL
LIN {X 0,Y 352.215,Z 331.743,A -85,B 0,C 180,E1 -13745.403,E2 -13745.403} C_VEL
LIN {X 0,Y 356.145,Z 351.363,A -85,B 0,C 180,E1 -13746.375,E2 -13746.375} C_VEL
LIN {X 0,Y 358.87,Z 370.781,A -85,B 0,C 180,E1 -13747.171,E2 -13747.171} C_VEL
LIN {X 0,Y 359.202,Z 377.618,A -85,B 0,C 180,E1 -13747.393,E2 -13747.393} C_VEL
LIN {X 0,Y 356.956,Z 443.876,A -85,B 0,C 180,E1 -13749.059,E2 -13749.059} C_VEL
LIN {X 0,Y 355.897,Z 458.074,A -85,B 0,C 180,E1 -13749.636,E2 -13749.636} C_VEL
LIN {X 0,Y 354.796,Z 469.745,A -85,B 0,C 180,E1 -13750.325,E2 -13750.325} C_VEL
LIN {X 0,Y 353.459,Z 482.154,A -85,B 0,C 180,E1 -13751.303,E2 -13751.303} C_VEL
LIN {X 0,Y 352.063,Z 493.391,A -85,B 0,C 180,E1 -13752.43,E2 -13752.43} C_VEL
LIN {X 0,Y 350.735,Z 503.603,A -85,B 0,C 180,E1 -13753.712,E2 -13753.712} C_VEL
LIN {X 0,Y 349.527,Z 512.89,A -85,B 0,C 180,E1 -13755.149,E2 -13755.149} C_VEL
LIN {X 0,Y 348.395,Z 522.006,A -85,B 0,C 180,E1 -13756.886,E2 -13756.886} C_VEL
LIN {X 0,Y 347.37,Z 529.377,A -85,B 0,C 180,E1 -13758.626,E2 -13758.626} C_VEL
LIN {X 0,Y 346.725,Z 536.154,A -85,B 0,C 180,E1 -13760.671,E2 -13760.671} C_VEL
LIN {X 0,Y 346.4,Z 540.655,A -85,B 0,C 180,E1 -13762.425,E2 -13762.425} C_VEL
LIN {X 0,Y 346.25,Z 544.055,A -85,B 0,C 180,E1 -13764.178,E2 -13764.178} C_VEL
LIN {X 0,Y 346.23,Z 545.772,A -85,B 0,C 180,E1 -13765.345,E2 -13765.345} C_VEL
LIN {X 0,Y 346.203,Z 547.037,A -85,B 0,C 180,E1 -13766.511,E2 -13766.511} C_VEL
LIN {X 0,Y 346.234,Z 547.856,A -85,B 0,C 180,E1 -13767.675,E2 -13767.675} C_VEL
LIN {X 0,Y 346.37,Z 548.274,A -85,B 0,C 180,E1 -13768.839,E2 -13768.839} C_VEL
LIN {X 0,Y 346.395,Z 548.279,A -85,B 0,C 180,E1 -13770.002,E2 -13770.002} C_VEL
LIN {X 0,Y 346.405,Z 547.828,A -85,B 0,C 180,E1 -13771.164,E2 -13771.164} C_VEL
LIN {X 0,Y 346.31,Z 546.932,A -85,B 0,C 180,E1 -13772.328,E2 -13772.328} C_VEL
LIN {X 0,Y 346.239,Z 545.616,A -85,B 0,C 180,E1 -13773.493,E2 -13773.493} C_VEL
LIN {X 0,Y 346.314,Z 542.778,A -85,B 0,C 180,E1 -13775.241,E2 -13775.241} C_VEL
LIN {X 0,Y 346.411,Z 538.84,A -85,B 0,C 180,E1 -13776.993,E2 -13776.993} C_VEL
LIN {X 0,Y 346.558,Z 533.697,A -85,B 0,C 180,E1 -13778.749,E2 -13778.749} C_VEL
LIN {X 0,Y 346.937,Z 527.188,A -85,B 0,C 180,E1 -13780.505,E2 -13780.505} C_VEL
LIN {X 0,Y 347.656,Z 519.014,A -85,B 0,C 180,E1 -13782.256,E2 -13782.256} C_VEL
LIN {X 0,Y 348.424,Z 510.668,A -85,B 0,C 180,E1 -13783.71,E2 -13783.71} C_VEL
LIN {X 0,Y 349.205,Z 500.447,A -85,B 0,C 180,E1 -13785.167,E2 -13785.167} C_VEL
LIN {X 0,Y 350.308,Z 488.929,A -85,B 0,C 180,E1 -13786.462,E2 -13786.462} C_VEL
LIN {X 0,Y 351.246,Z 477.679,A -85,B 0,C 180,E1 -13787.466,E2 -13787.466} C_VEL
LIN {X 0,Y 352.064,Z 466.385,A -85,B 0,C 180,E1 -13788.25,E2 -13788.25} C_VEL
LIN {X 0,Y 352.871,Z 452.974,A -85,B 0,C 180,E1 -13788.921,E2 -13788.921} C_VEL
LIN {X 0,Y 353.428,Z 440.016,A -85,B 0,C 180,E1 -13789.342,E2 -13789.342} C_VEL
LIN {X 0,Y 354.776,Z 373.279,A -85,B 0,C 180,E1 -13790.914,E2 -13790.914} C_VEL
LIN {X 0,Y 350.073,Z 336.371,A -85,B 0,C 180,E1 -13792.073,E2 -13792.073} C_VEL
LIN {X 0,Y 351.825,Z 318.798,A -85,B 0,C 180,E1 -13795.984,E2 -13795.984} C_VEL
LIN {X 0,Y 351.249,Z 314.193,A -85,B 0,C 180,E1 -13797.077,E2 -13797.077} C_VEL
LIN {X 0,Y 348.899,Z 302.376,A -85,B 0,C 180,E1 -13799.983,E2 -13799.983} C_VEL
LIN {X 0,Y 347.766,Z 297.166,A -85,B 0,C 180,E1 -13801.356,E2 -13801.356} C_VEL
LIN {X 0,Y 347.739,Z 297.17,A -85,B 0,C 180,E1 -13804.463,E2 -13804.463} C_VEL
LIN {X 0,Y 347.756,Z 297.164,A -85,B 0,C 180,E1 -13807.984,E2 -13807.984} C_VEL
LIN {X 0,Y 347.732,Z 297.167,A -85,B 0,C 180,E1 -13811.83,E2 -13811.83} C_VEL
LIN {X 0,Y 347.689,Z 297.176,A -85,B 0,C 180,E1 -13815.026,E2 -13815.026} C_VEL
LIN {X 0,Y 347.698,Z 297.172,A -85,B 0,C 180,E1 -13818.403,E2 -13818.403} C_VEL
LIN {X 0,Y 347.748,Z 297.165,A -85,B 0,C 180,E1 -13822.012,E2 -13822.012} C_VEL
LIN {X 0,Y 347.728,Z 297.169,A -85,B 0,C 180,E1 -13825.534,E2 -13825.534} C_VEL
LIN {X 0,Y 347.716,Z 297.17,A -85,B 0,C 180,E1 -13829.648,E2 -13829.648} C_VEL
LIN {X 0,Y 347.746,Z 297.168,A -85,B 0,C 180,E1 -13832.771,E2 -13832.771} C_VEL
LIN {X 0,Y 347.743,Z 297.166,A -85,B 0,C 180,E1 -13836.158,E2 -13836.158} C_VEL
LIN {X 0,Y 347.757,Z 297.164,A -85,B 0,C 180,E1 -13839.905,E2 -13839.905} C_VEL
LIN {X 0,Y 347.82,Z 297.156,A -85,B 0,C 180,E1 -13842.356,E2 -13842.356} C_VEL
LIN {X 0,Y 347.877,Z 297.15,A -85,B 0,C 180,E1 -13845.969,E2 -13845.969} C_VEL
LIN {X 0,Y 347.873,Z 297.154,A -85,B 0,C 180,E1 -13849.523,E2 -13849.523} C_VEL
LIN {X 0,Y 348.063,Z 297.129,A -85,B 0,C 180,E1 -13853.041,E2 -13853.041} C_VEL
LIN {X 0,Y 348.175,Z 297.116,A -85,B 0,C 180,E1 -13857.686,E2 -13857.686} C_VEL
LIN {X 0,Y 348.259,Z 297.103,A -85,B 0,C 180,E1 -13859.999,E2 -13859.999} C_VEL
LIN {X 0,Y 348.175,Z 297.112,A -85,B 0,C 180,E1 -13862.313,E2 -13862.313} C_VEL
LIN {X 0,Y 348.061,Z 297.127,A -85,B 0,C 180,E1 -13866.958,E2 -13866.958} C_VEL
LIN {X 0,Y 347.905,Z 297.146,A -85,B 0,C 180,E1 -13870.475,E2 -13870.475} C_VEL
LIN {X 0,Y 347.876,Z 297.151,A -85,B 0,C 180,E1 -13874.15,E2 -13874.15} C_VEL
LIN {X 0,Y 347.786,Z 297.162,A -85,B 0,C 180,E1 -13878.249,E2 -13878.249} C_VEL
LIN {X 0,Y 347.745,Z 297.171,A -85,B 0,C 180,E1 -13881.626,E2 -13881.626} C_VEL
LIN {X 0,Y 347.789,Z 297.161,A -85,B 0,C 180,E1 -13885.11,E2 -13885.11} C_VEL
LIN {X 0,Y 347.79,Z 297.165,A -85,B 0,C 180,E1 -13887.695,E2 -13887.695} C_VEL
LIN {X 0,Y 347.744,Z 297.167,A -85,B 0,C 180,E1 -13890.348,E2 -13890.348} C_VEL
LIN {X 0,Y 347.726,Z 297.169,A -85,B 0,C 180,E1 -13894.465,E2 -13894.465} C_VEL
LIN {X 0,Y 347.758,Z 297.169,A -85,B 0,C 180,E1 -13897.99,E2 -13897.99} C_VEL
LIN {X 0,Y 347.744,Z 297.17,A -85,B 0,C 180,E1 -13901.83,E2 -13901.83} C_VEL
LIN {X 0,Y 347.763,Z 297.163,A -85,B 0,C 180,E1 -13905.016,E2 -13905.016} C_VEL
LIN {X 0,Y 347.772,Z 297.166,A -85,B 0,C 180,E1 -13908.392,E2 -13908.392} C_VEL
LIN {X 0,Y 347.768,Z 297.167,A -85,B 0,C 180,E1 -13912.012,E2 -13912.012} C_VEL
LIN {X 0,Y 347.736,Z 297.167,A -85,B 0,C 180,E1 -13915.537,E2 -13915.537} C_VEL
LIN {X 0,Y 347.737,Z 297.172,A -85,B 0,C 180,E1 -13918.301,E2 -13918.301} C_VEL
LIN {X 0,Y 347.772,Z 297.163,A -85,B 0,C 180,E1 -13920.988,E2 -13920.988} C_VEL
LIN {X 0,Y 347.825,Z 297.156,A -85,B 0,C 180,E1 -13923.608,E2 -13923.608} C_VEL
LIN {X 0,Y 347.784,Z 297.165,A -85,B 0,C 180,E1 -13926.162,E2 -13926.162} C_VEL
LIN {X 0,Y 347.814,Z 297.159,A -85,B 0,C 180,E1 -13929.91,E2 -13929.91} C_VEL
LIN {X 0,Y 347.863,Z 297.155,A -85,B 0,C 180,E1 -13932.359,E2 -13932.359} C_VEL
LIN {X 0,Y 347.895,Z 297.148,A -85,B 0,C 180,E1 -13935.97,E2 -13935.97} C_VEL
LIN {X 0,Y 347.926,Z 297.143,A -85,B 0,C 180,E1 -13939.525,E2 -13939.525} C_VEL
LIN {X 0,Y 348.072,Z 297.125,A -85,B 0,C 180,E1 -13941.874,E2 -13941.874} C_VEL
LIN {X 0,Y 348.065,Z 297.128,A -85,B 0,C 180,E1 -13944.204,E2 -13944.204} C_VEL
LIN {X 0,Y 348.205,Z 297.108,A -85,B 0,C 180,E1 -13947.685,E2 -13947.685} C_VEL
LIN {X 0,Y 348.343,Z 297.092,A -85,B 0,C 180,E1 -13949.998,E2 -13949.998} C_VEL
LIN {X 0,Y 348.205,Z 297.111,A -85,B 0,C 180,E1 -13952.311,E2 -13952.311} C_VEL
LIN {X 0,Y 348.099,Z 297.125,A -85,B 0,C 180,E1 -13956.955,E2 -13956.955} C_VEL
LIN {X 0,Y 347.925,Z 297.146,A -85,B 0,C 180,E1 -13960.472,E2 -13960.472} C_VEL
LIN {X 0,Y 347.89,Z 297.148,A -85,B 0,C 180,E1 -13964.147,E2 -13964.147} C_VEL
LIN {X 0,Y 347.882,Z 297.149,A -85,B 0,C 180,E1 -13968.288,E2 -13968.288} C_VEL
LIN {X 0,Y 347.801,Z 297.159,A -85,B 0,C 180,E1 -13971.642,E2 -13971.642} C_VEL
LIN {X 0,Y 347.803,Z 297.163,A -85,B 0,C 180,E1 -13975.104,E2 -13975.104} C_VEL
LIN {X 0,Y 347.796,Z 297.159,A -85,B 0,C 180,E1 -13977.69,E2 -13977.69} C_VEL
LIN {X 0,Y 347.747,Z 297.165,A -85,B 0,C 180,E1 -13980.343,E2 -13980.343} C_VEL
LIN {X 0,Y 347.723,Z 297.168,A -85,B 0,C 180,E1 -13984.46,E2 -13984.46} C_VEL
LIN {X 0,Y 347.756,Z 297.166,A -85,B 0,C 180,E1 -13987.986,E2 -13987.986} C_VEL
LIN {X 0,Y 347.808,Z 297.168,A -85,B 0,C 180,E1 -13989.544,E2 -13989.544} C_VEL
LIN {X 0,Y 348.139,Z 298.791,A -85,B 0,C 180,E1 -13989.943,E2 -13989.943} C_VEL
LIN {X 0,Y 355.008,Z 320.024,A -85,B 0,C 180,E1 -13990.83,E2 -13990.83} C_VEL
LIN {X 0,Y 355.56,Z 323.301,A -85,B 0,C 180,E1 -13990.939,E2 -13990.939} C_VEL
LIN {X 0,Y 353.5,Z 407.12,A -85,B 0,C 180,E1 -13992.931,E2 -13992.931} C_VEL
LIN {X 0,Y 353.239,Z 414.124,A -85,B 0,C 180,E1 -13993.19,E2 -13993.19} C_VEL
LIN {X 0,Y 352.432,Z 419.807,A -85,B 0,C 180,E1 -13993.421,E2 -13993.421} C_VEL
LIN {X 0,Y 349.181,Z 428.885,A -85,B 0,C 180,E1 -13993.813,E2 -13993.813} C_VEL
LIN {X 0,Y 345.815,Z 437.697,A -85,B 0,C 180,E1 -13994.322,E2 -13994.322} C_VEL
LIN {X 0,Y 344.837,Z 442.962,A -85,B 0,C 180,E1 -13994.736,E2 -13994.736} C_VEL
LIN {X 0,Y 343.99,Z 453.795,A -85,B 0,C 180,E1 -13995.799,E2 -13995.799} C_VEL
LIN {X 0,Y 343.095,Z 464.211,A -85,B 0,C 180,E1 -13997.072,E2 -13997.072} C_VEL
LIN {X 0,Y 342.212,Z 473.887,A -85,B 0,C 180,E1 -13998.524,E2 -13998.524} C_VEL
LIN {X 0,Y 341.51,Z 481.615,A -85,B 0,C 180,E1 -13999.938,E2 -13999.938} C_VEL
LIN {X 0,Y 340.701,Z 489.754,A -85,B 0,C 180,E1 -14001.769,E2 -14001.769} C_VEL
LIN {X 0,Y 340.146,Z 496.465,A -85,B 0,C 180,E1 -14003.677,E2 -14003.677} C_VEL
LIN {X 0,Y 339.778,Z 500.924,A -85,B 0,C 180,E1 -14005.276,E2 -14005.276} C_VEL
LIN {X 0,Y 339.431,Z 505.498,A -85,B 0,C 180,E1 -14007.43,E2 -14007.43} C_VEL
LIN {X 0,Y 339.213,Z 507.571,A -85,B 0,C 180,E1 -14008.805,E2 -14008.805} C_VEL
LIN {X 0,Y 339.085,Z 509.358,A -85,B 0,C 180,E1 -14010.503,E2 -14010.503} C_VEL
LIN {X 0,Y 339.1,Z 510.432,A -85,B 0,C 180,E1 -14012.874,E2 -14012.874} C_VEL
LIN {X 0,Y 339.192,Z 510.282,A -85,B 0,C 180,E1 -14014.208,E2 -14014.208} C_VEL
LIN {X 0,Y 339.4,Z 509.562,A -85,B 0,C 180,E1 -14015.642,E2 -14015.642} C_VEL
LIN {X 0,Y 339.618,Z 508.48,A -85,B 0,C 180,E1 -14016.848,E2 -14016.848} C_VEL
LIN {X 0,Y 340.042,Z 506.396,A -85,B 0,C 180,E1 -14018.425,E2 -14018.425} C_VEL
LIN {X 0,Y 340.509,Z 503.33,A -85,B 0,C 180,E1 -14020.09,E2 -14020.09} C_VEL
LIN {X 0,Y 341.285,Z 498.621,A -85,B 0,C 180,E1 -14022.008,E2 -14022.008} C_VEL
LIN {X 0,Y 342.271,Z 492.492,A -85,B 0,C 180,E1 -14023.908,E2 -14023.908} C_VEL
LIN {X 0,Y 343.539,Z 484.724,A -85,B 0,C 180,E1 -14025.79,E2 -14025.79} C_VEL
LIN {X 0,Y 344.884,Z 475.849,A -85,B 0,C 180,E1 -14027.501,E2 -14027.501} C_VEL
LIN {X 0,Y 346.307,Z 465.882,A -85,B 0,C 180,E1 -14029.033,E2 -14029.033} C_VEL
LIN {X 0,Y 347.768,Z 454.758,A -85,B 0,C 180,E1 -14030.403,E2 -14030.403} C_VEL
LIN {X 0,Y 349.003,Z 442.791,A -85,B 0,C 180,E1 -14031.559,E2 -14031.559} C_VEL
LIN {X 0,Y 350.148,Z 429.981,A -85,B 0,C 180,E1 -14032.504,E2 -14032.504} C_VEL
LIN {X 0,Y 351.002,Z 416.589,A -85,B 0,C 180,E1 -14033.209,E2 -14033.209} C_VEL
LIN {X 0,Y 351.574,Z 403.786,A -85,B 0,C 180,E1 -14033.652,E2 -14033.652} C_VEL
LIN {X 0,Y 354.399,Z 327.479,A -85,B 0,C 180,E1 -14035.601,E2 -14035.601} C_VEL
LIN {X 0,Y 349.927,Z 316.933,A -85,B 0,C 180,E1 -14036.376,E2 -14036.376} C_VEL
LIN {X 0,Y 341.951,Z 301.002,A -85,B 0,C 180,E1 -14037.792,E2 -14037.792} C_VEL
LIN {X 0,Y 341.077,Z 298.002,A -85,B 0,C 180,E1 -14038.672,E2 -14038.672} C_VEL
LIN {X 0,Y 341.227,Z 297.981,A -85,B 0,C 180,E1 -14040.001,E2 -14040.001} C_VEL
LIN {X 0,Y 341.121,Z 297.995,A -85,B 0,C 180,E1 -14042.362,E2 -14042.362} C_VEL
LIN {X 0,Y 341.011,Z 298.01,A -85,B 0,C 180,E1 -14047.104,E2 -14047.104} C_VEL
LIN {X 0,Y 340.827,Z 298.028,A -85,B 0,C 180,E1 -14050.696,E2 -14050.696} C_VEL
LIN {X 0,Y 340.821,Z 298.031,A -85,B 0,C 180,E1 -14054.327,E2 -14054.327} C_VEL
LIN {X 0,Y 340.742,Z 298.037,A -85,B 0,C 180,E1 -14058.442,E2 -14058.442} C_VEL
LIN {X 0,Y 340.679,Z 298.047,A -85,B 0,C 180,E1 -14061.845,E2 -14061.845} C_VEL
LIN {X 0,Y 340.733,Z 298.036,A -85,B 0,C 180,E1 -14065.668,E2 -14065.668} C_VEL
LIN {X 0,Y 340.682,Z 298.046,A -85,B 0,C 180,E1 -14068.326,E2 -14068.326} C_VEL
LIN {X 0,Y 340.657,Z 298.049,A -85,B 0,C 180,E1 -14071.049,E2 -14071.049} C_VEL
LIN {X 0,Y 340.686,Z 298.046,A -85,B 0,C 180,E1 -14075.283,E2 -14075.283} C_VEL
LIN {X 0,Y 340.683,Z 298.047,A -85,B 0,C 180,E1 -14078.391,E2 -14078.391} C_VEL
LIN {X 0,Y 340.679,Z 298.044,A -85,B 0,C 180,E1 -14082.051,E2 -14082.051} C_VEL
LIN {X 0,Y 340.628,Z 298.054,A -85,B 0,C 180,E1 -14086.232,E2 -14086.232} C_VEL
LIN {X 0,Y 340.667,Z 298.051,A -85,B 0,C 180,E1 -14089.758,E2 -14089.758} C_VEL
LIN {X 0,Y 340.686,Z 298.05,A -85,B 0,C 180,E1 -14093.263,E2 -14093.263} C_VEL
LIN {X 0,Y 340.678,Z 298.057,A -85,B 0,C 180,E1 -14096.336,E2 -14096.336} C_VEL
LIN {X 0,Y 343.608,Z 308.437,A -85,B 0,C 180,E1 -14099.253,E2 -14099.253} C_VEL
LIN {X 0,Y 345.91,Z 318.702,A -85,B 0,C 180,E1 -14101.902,E2 -14101.902} C_VEL
LIN {X 0,Y 346.557,Z 323.944,A -85,B 0,C 180,E1 -14103.164,E2 -14103.164} C_VEL
LIN {X 0,Y 345.685,Z 331.283,A -85,B 0,C 180,E1 -14104.731,E2 -14104.731} C_VEL
LIN {X 0,Y 349.571,Z 350.492,A -85,B 0,C 180,E1 -14105.719,E2 -14105.719} C_VEL
LIN {X 0,Y 352.212,Z 368.091,A -85,B 0,C 180,E1 -14106.501,E2 -14106.501} C_VEL
LIN {X 0,Y 352.96,Z 377.798,A -85,B 0,C 180,E1 -14106.851,E2 -14106.851} C_VEL
LIN {X 0,Y 350.607,Z 443.671,A -85,B 0,C 180,E1 -14108.546,E2 -14108.546} C_VEL
LIN {X 0,Y 349.575,Z 456.959,A -85,B 0,C 180,E1 -14109.097,E2 -14109.097} C_VEL
LIN {X 0,Y 348.386,Z 468.764,A -85,B 0,C 180,E1 -14109.794,E2 -14109.794} C_VEL
LIN {X 0,Y 346.977,Z 481.216,A -85,B 0,C 180,E1 -14110.787,E2 -14110.787} C_VEL
LIN {X 0,Y 345.496,Z 492.503,A -85,B 0,C 180,E1 -14111.932,E2 -14111.932} C_VEL
LIN {X 0,Y 344.085,Z 502.825,A -85,B 0,C 180,E1 -14113.235,E2 -14113.235} C_VEL
LIN {X 0,Y 342.665,Z 513.017,A -85,B 0,C 180,E1 -14114.845,E2 -14114.845} C_VEL
LIN {X 0,Y 341.468,Z 522.048,A -85,B 0,C 180,E1 -14116.615,E2 -14116.615} C_VEL
LIN {X 0,Y 340.391,Z 529.296,A -85,B 0,C 180,E1 -14118.39,E2 -14118.39} C_VEL
LIN {X 0,Y 339.687,Z 535.989,A -85,B 0,C 180,E1 -14120.476,E2 -14120.476} C_VEL
LIN {X 0,Y 339.342,Z 540.428,A -85,B 0,C 180,E1 -14122.266,E2 -14122.266} C_VEL
LIN {X 0,Y 339.17,Z 543.781,A -85,B 0,C 180,E1 -14124.056,E2 -14124.056} C_VEL
LIN {X 0,Y 339.128,Z 545.472,A -85,B 0,C 180,E1 -14125.247,E2 -14125.247} C_VEL
LIN {X 0,Y 339.125,Z 546.689,A -85,B 0,C 180,E1 -14126.438,E2 -14126.438} C_VEL
LIN {X 0,Y 339.288,Z 547.879,A -85,B 0,C 180,E1 -14128.815,E2 -14128.815} C_VEL
LIN {X 0,Y 339.333,Z 547.85,A -85,B 0,C 180,E1 -14130.002,E2 -14130.002} C_VEL
LIN {X 0,Y 339.341,Z 547.353,A -85,B 0,C 180,E1 -14131.188,E2 -14131.188} C_VEL
LIN {X 0,Y 339.216,Z 546.426,A -85,B 0,C 180,E1 -14132.376,E2 -14132.376} C_VEL
LIN {X 0,Y 339.165,Z 545.082,A -85,B 0,C 180,E1 -14133.566,E2 -14133.566} C_VEL
LIN {X 0,Y 339.251,Z 543.273,A -85,B 0,C 180,E1 -14134.755,E2 -14134.755} C_VEL
LIN {X 0,Y 339.318,Z 539.791,A -85,B 0,C 180,E1 -14136.483,E2 -14136.483} C_VEL
LIN {X 0,Y 339.424,Z 534.827,A -85,B 0,C 180,E1 -14138.335,E2 -14138.335} C_VEL
LIN {X 0,Y 339.773,Z 528.693,A -85,B 0,C 180,E1 -14140.127,E2 -14140.127} C_VEL
LIN {X 0,Y 340.412,Z 521.032,A -85,B 0,C 180,E1 -14141.915,E2 -14141.915} C_VEL
LIN {X 0,Y 341.066,Z 513.186,A -85,B 0,C 180,E1 -14143.405,E2 -14143.405} C_VEL
LIN {X 0,Y 341.83,Z 504.529,A -85,B 0,C 180,E1 -14144.762,E2 -14144.762} C_VEL
LIN {X 0,Y 342.893,Z 492.98,A -85,B 0,C 180,E1 -14146.216,E2 -14146.216} C_VEL
LIN {X 0,Y 343.96,Z 481.219,A -85,B 0,C 180,E1 -14147.387,E2 -14147.387} C_VEL
LIN {X 0,Y 344.901,Z 468.752,A -85,B 0,C 180,E1 -14148.335,E2 -14148.335} C_VEL
LIN {X 0,Y 345.869,Z 455.178,A -85,B 0,C 180,E1 -14149.088,E2 -14149.088} C_VEL
LIN {X 0,Y 346.451,Z 442.38,A -85,B 0,C 180,E1 -14149.555,E2 -14149.555} C_VEL
LIN {X 0,Y 347.885,Z 373.581,A -85,B 0,C 180,E1 -14151.229,E2 -14151.229} C_VEL
LIN {X 0,Y 343.129,Z 335.966,A -85,B 0,C 180,E1 -14152.456,E2 -14152.456} C_VEL
LIN {X 0,Y 344.714,Z 321.138,A -85,B 0,C 180,E1 -14155.816,E2 -14155.816} C_VEL
LIN {X 0,Y 344.676,Z 317.567,A -85,B 0,C 180,E1 -14156.652,E2 -14156.652} C_VEL
LIN {X 0,Y 342.15,Z 304.65,A -85,B 0,C 180,E1 -14159.886,E2 -14159.886} C_VEL
LIN {X 0,Y 340.705,Z 298.046,A -85,B 0,C 180,E1 -14161.648,E2 -14161.648} C_VEL
LIN {X 0,Y 340.711,Z 298.042,A -85,B 0,C 180,E1 -14165.278,E2 -14165.278} C_VEL
LIN {X 0,Y 340.687,Z 298.046,A -85,B 0,C 180,E1 -14168.38,E2 -14168.38} C_VEL
LIN {X 0,Y 340.683,Z 298.045,A -85,B 0,C 180,E1 -14172.042,E2 -14172.042} C_VEL
LIN {X 0,Y 340.639,Z 298.051,A -85,B 0,C 180,E1 -14176.226,E2 -14176.226} C_VEL
LIN {X 0,Y 340.639,Z 298.05,A -85,B 0,C 180,E1 -14179.759,E2 -14179.759} C_VEL
LIN {X 0,Y 340.687,Z 298.048,A -85,B 0,C 180,E1 -14183.255,E2 -14183.255} C_VEL
LIN {X 0,Y 340.675,Z 298.046,A -85,B 0,C 180,E1 -14186.151,E2 -14186.151} C_VEL
LIN {X 0,Y 340.709,Z 298.042,A -85,B 0,C 180,E1 -14190.326,E2 -14190.326} C_VEL
LIN {X 0,Y 340.705,Z 298.042,A -85,B 0,C 180,E1 -14194.33,E2 -14194.33} C_VEL
LIN {X 0,Y 340.705,Z 298.042,A -85,B 0,C 180,E1 -14198.204,E2 -14198.204} C_VEL
LIN {X 0,Y 340.77,Z 298.034,A -85,B 0,C 180,E1 -14201.979,E2 -14201.979} C_VEL
LIN {X 0,Y 340.832,Z 298.028,A -85,B 0,C 180,E1 -14205.715,E2 -14205.715} C_VEL
LIN {X 0,Y 340.825,Z 298.033,A -85,B 0,C 180,E1 -14209.304,E2 -14209.304} C_VEL
LIN {X 0,Y 341.032,Z 298.003,A -85,B 0,C 180,E1 -14212.897,E2 -14212.897} C_VEL
LIN {X 0,Y 341.137,Z 297.993,A -85,B 0,C 180,E1 -14217.638,E2 -14217.638} C_VEL
LIN {X 0,Y 341.211,Z 297.981,A -85,B 0,C 180,E1 -14219.999,E2 -14219.999} C_VEL
LIN {X 0,Y 341.137,Z 297.988,A -85,B 0,C 180,E1 -14222.361,E2 -14222.361} C_VEL
LIN {X 0,Y 341.03,Z 298.004,A -85,B 0,C 180,E1 -14227.102,E2 -14227.102} C_VEL
LIN {X 0,Y 340.847,Z 298.025,A -85,B 0,C 180,E1 -14230.694,E2 -14230.694} C_VEL
LIN {X 0,Y 340.841,Z 298.026,A -85,B 0,C 180,E1 -14234.325,E2 -14234.325} C_VEL
LIN {X 0,Y 340.747,Z 298.038,A -85,B 0,C 180,E1 -14238.432,E2 -14238.432} C_VEL
LIN {X 0,Y 340.697,Z 298.048,A -85,B 0,C 180,E1 -14241.842,E2 -14241.842} C_VEL
LIN {X 0,Y 340.75,Z 298.042,A -85,B 0,C 180,E1 -14245.665,E2 -14245.665} C_VEL
LIN {X 0,Y 340.721,Z 298.042,A -85,B 0,C 180,E1 -14248.321,E2 -14248.321} C_VEL
LIN {X 0,Y 340.685,Z 298.045,A -85,B 0,C 180,E1 -14251.045,E2 -14251.045} C_VEL
LIN {X 0,Y 340.7,Z 298.044,A -85,B 0,C 180,E1 -14255.28,E2 -14255.28} C_VEL
LIN {X 0,Y 340.696,Z 298.046,A -85,B 0,C 180,E1 -14258.387,E2 -14258.387} C_VEL
LIN {X 0,Y 340.691,Z 298.049,A -85,B 0,C 180,E1 -14262.048,E2 -14262.048} C_VEL
LIN {X 0,Y 340.7,Z 298.048,A -85,B 0,C 180,E1 -14266.218,E2 -14266.218} C_VEL
LIN {X 0,Y 340.753,Z 298.039,A -85,B 0,C 180,E1 -14269.739,E2 -14269.739} C_VEL
LIN {X 0,Y 340.702,Z 298.044,A -85,B 0,C 180,E1 -14273.56,E2 -14273.56} C_VEL
LIN {X 0,Y 340.684,Z 298.05,A -85,B 0,C 180,E1 -14276.154,E2 -14276.154} C_VEL
LIN {X 0,Y 340.735,Z 298.044,A -85,B 0,C 180,E1 -14280.33,E2 -14280.33} C_VEL
LIN {X 0,Y 340.798,Z 298.031,A -85,B 0,C 180,E1 -14283.02,E2 -14283.02} C_VEL
LIN {X 0,Y 340.724,Z 298.041,A -85,B 0,C 180,E1 -14286.927,E2 -14286.927} C_VEL
LIN {X 0,Y 340.791,Z 298.034,A -85,B 0,C 180,E1 -14290.734,E2 -14290.734} C_VEL
LIN {X 0,Y 340.783,Z 298.033,A -85,B 0,C 180,E1 -14293.218,E2 -14293.218} C_VEL
LIN {X 0,Y 340.842,Z 298.027,A -85,B 0,C 180,E1 -14296.89,E2 -14296.89} C_VEL
LIN {X 0,Y 340.926,Z 298.02,A -85,B 0,C 180,E1 -14300.507,E2 -14300.507} C_VEL
LIN {X 0,Y 341.074,Z 297.999,A -85,B 0,C 180,E1 -14302.897,E2 -14302.897} C_VEL
LIN {X 0,Y 341.167,Z 297.985,A -85,B 0,C 180,E1 -14307.637,E2 -14307.637} C_VEL
LIN {X 0,Y 341.294,Z 297.97,A -85,B 0,C 180,E1 -14309.998,E2 -14309.998} C_VEL
LIN {X 0,Y 341.167,Z 297.988,A -85,B 0,C 180,E1 -14312.359,E2 -14312.359} C_VEL
LIN {X 0,Y 341.069,Z 297.999,A -85,B 0,C 180,E1 -14317.099,E2 -14317.099} C_VEL
LIN {X 0,Y 340.868,Z 298.027,A -85,B 0,C 180,E1 -14320.691,E2 -14320.691} C_VEL
LIN {X 0,Y 340.855,Z 298.025,A -85,B 0,C 180,E1 -14324.322,E2 -14324.322} C_VEL
LIN {X 0,Y 340.829,Z 298.029,A -85,B 0,C 180,E1 -14328.464,E2 -14328.464} C_VEL
LIN {X 0,Y 340.742,Z 298.037,A -85,B 0,C 180,E1 -14331.853,E2 -14331.853} C_VEL
LIN {X 0,Y 340.761,Z 298.036,A -85,B 0,C 180,E1 -14335.66,E2 -14335.66} C_VEL
LIN {X 0,Y 340.726,Z 298.04,A -85,B 0,C 180,E1 -14338.316,E2 -14338.316} C_VEL
LIN {X 0,Y 340.686,Z 298.05,A -85,B 0,C 180,E1 -14341.04,E2 -14341.04} C_VEL
LIN {X 0,Y 340.697,Z 298.047,A -85,B 0,C 180,E1 -14345.275,E2 -14345.275} C_VEL
LIN {X 0,Y 340.806,Z 298.231,A -85,B 0,C 180,E1 -14349.363,E2 -14349.363} C_VEL
LIN {X 0,Y 340.991,Z 299.168,A -85,B 0,C 180,E1 -14349.567,E2 -14349.567} C_VEL
LIN {X 0,Y 348.43,Z 322.018,A -85,B 0,C 180,E1 -14350.554,E2 -14350.554} C_VEL
LIN {X 0,Y 348.724,Z 325.633,A -85,B 0,C 180,E1 -14350.661,E2 -14350.661} C_VEL
LIN {X 0,Y 346.626,Z 407.157,A -85,B 0,C 180,E1 -14352.641,E2 -14352.641} C_VEL
LIN {X 0,Y 346.184,Z 420.034,A -85,B 0,C 180,E1 -14353.178,E2 -14353.178} C_VEL
LIN {X 0,Y 345.521,Z 432.429,A -85,B 0,C 180,E1 -14353.912,E2 -14353.912} C_VEL
LIN {X 0,Y 344.837,Z 442.962,A -85,B 0,C 180,E1 -14354.736,E2 -14354.736} C_VEL
LIN {X 0,Y 343.858,Z 448.145,A -85,B 0,C 180,E1 -14355.189,E2 -14355.189} C_VEL
LIN {X 0,Y 340.411,Z 456.247,A -85,B 0,C 180,E1 -14355.943,E2 -14355.943} C_VEL
LIN {X 0,Y 336.884,Z 463.977,A -85,B 0,C 180,E1 -14356.809,E2 -14356.809} C_VEL
LIN {X 0,Y 335.792,Z 468.482,A -85,B 0,C 180,E1 -14357.433,E2 -14357.433} C_VEL
LIN {X 0,Y 334.837,Z 478.292,A -85,B 0,C 180,E1 -14359.07,E2 -14359.07} C_VEL
LIN {X 0,Y 333.956,Z 486.834,A -85,B 0,C 180,E1 -14360.852,E2 -14360.852} C_VEL
LIN {X 0,Y 333.289,Z 494.428,A -85,B 0,C 180,E1 -14362.846,E2 -14362.846} C_VEL
LIN {X 0,Y 332.842,Z 499.436,A -85,B 0,C 180,E1 -14364.503,E2 -14364.503} C_VEL
LIN {X 0,Y 332.482,Z 504.462,A -85,B 0,C 180,E1 -14366.662,E2 -14366.662} C_VEL
LIN {X 0,Y 332.201,Z 506.904,A -85,B 0,C 180,E1 -14368.07,E2 -14368.07} C_VEL
LIN {X 0,Y 331.998,Z 509.482,A -85,B 0,C 180,E1 -14370.204,E2 -14370.204} C_VEL
LIN {X 0,Y 332.001,Z 510.796,A -85,B 0,C 180,E1 -14372.742,E2 -14372.742} C_VEL
LIN {X 0,Y 332.201,Z 510.499,A -85,B 0,C 180,E1 -14374.969,E2 -14374.969} C_VEL
LIN {X 0,Y 332.43,Z 509.602,A -85,B 0,C 180,E1 -14376.317,E2 -14376.317} C_VEL
LIN {X 0,Y 332.9,Z 507.439,A -85,B 0,C 180,E1 -14378.245,E2 -14378.245} C_VEL
LIN {X 0,Y 333.529,Z 503.906,A -85,B 0,C 180,E1 -14380.298,E2 -14380.298} C_VEL
LIN {X 0,Y 334.349,Z 499.239,A -85,B 0,C 180,E1 -14382.255,E2 -14382.255} C_VEL
LIN {X 0,Y 335.399,Z 493.171,A -85,B 0,C 180,E1 -14384.193,E2 -14384.193} C_VEL
LIN {X 0,Y 336.746,Z 485.475,A -85,B 0,C 180,E1 -14386.114,E2 -14386.114} C_VEL
LIN {X 0,Y 338.029,Z 477.579,A -85,B 0,C 180,E1 -14387.701,E2 -14387.701} C_VEL
LIN {X 0,Y 339.518,Z 467.958,A -85,B 0,C 180,E1 -14389.264,E2 -14389.264} C_VEL
LIN {X 0,Y 341.086,Z 456.817,A -85,B 0,C 180,E1 -14390.7,E2 -14390.7} C_VEL
LIN {X 0,Y 342.406,Z 445.22,A -85,B 0,C 180,E1 -14391.888,E2 -14391.888} C_VEL
LIN {X 0,Y 343.634,Z 432.522,A -85,B 0,C 180,E1 -14392.878,E2 -14392.878} C_VEL
LIN {X 0,Y 344.507,Z 419.527,A -85,B 0,C 180,E1 -14393.632,E2 -14393.632} C_VEL
LIN {X 0,Y 345.25,Z 405.463,A -85,B 0,C 180,E1 -14394.159,E2 -14394.159} C_VEL
LIN {X 0,Y 348.244,Z 329.252,A -85,B 0,C 180,E1 -14396.168,E2 -14396.168} C_VEL
LIN {X 0,Y 343.423,Z 318.354,A -85,B 0,C 180,E1 -14397.022,E2 -14397.022} C_VEL
LIN {X 0,Y 335.985,Z 303.932,A -85,B 0,C 180,E1 -14398.372,E2 -14398.372} C_VEL
LIN {X 0,Y 334.866,Z 301.698,A -85,B 0,C 180,E1 -14398.61,E2 -14398.61} C_VEL
LIN {X 0,Y 334.102,Z 298.87,A -85,B 0,C 180,E1 -14399.473,E2 -14399.473} C_VEL
LIN {X 0,Y 334.059,Z 298.874,A -85,B 0,C 180,E1 -14402.412,E2 -14402.412} C_VEL
LIN {X 0,Y 333.966,Z 298.884,A -85,B 0,C 180,E1 -14406.04,E2 -14406.04} C_VEL
LIN {X 0,Y 333.806,Z 298.904,A -85,B 0,C 180,E1 -14409.697,E2 -14409.697} C_VEL
LIN {X 0,Y 333.75,Z 298.911,A -85,B 0,C 180,E1 -14413.394,E2 -14413.394} C_VEL
LIN {X 0,Y 333.674,Z 298.917,A -85,B 0,C 180,E1 -14417.151,E2 -14417.151} C_VEL
LIN {X 0,Y 333.619,Z 298.923,A -85,B 0,C 180,E1 -14419.698,E2 -14419.698} C_VEL
LIN {X 0,Y 333.63,Z 298.923,A -85,B 0,C 180,E1 -14423.594,E2 -14423.594} C_VEL
LIN {X 0,Y 333.692,Z 298.913,A -85,B 0,C 180,E1 -14426.251,E2 -14426.251} C_VEL
LIN {X 0,Y 333.643,Z 298.92,A -85,B 0,C 180,E1 -14428.979,E2 -14428.979} C_VEL
LIN {X 0,Y 333.603,Z 298.931,A -85,B 0,C 180,E1 -14433.213,E2 -14433.213} C_VEL
LIN {X 0,Y 333.645,Z 298.923,A -85,B 0,C 180,E1 -14436.144,E2 -14436.144} C_VEL
LIN {X 0,Y 333.641,Z 298.923,A -85,B 0,C 180,E1 -14439.194,E2 -14439.194} C_VEL
LIN {X 0,Y 333.611,Z 298.924,A -85,B 0,C 180,E1 -14442.505,E2 -14442.505} C_VEL
LIN {X 0,Y 333.572,Z 298.934,A -85,B 0,C 180,E1 -14445.959,E2 -14445.959} C_VEL
LIN {X 0,Y 333.627,Z 298.928,A -85,B 0,C 180,E1 -14449.32,E2 -14449.32} C_VEL
LIN {X 0,Y 333.647,Z 298.927,A -85,B 0,C 180,E1 -14453.173,E2 -14453.173} C_VEL
LIN {X 0,Y 333.694,Z 299.131,A -85,B 0,C 180,E1 -14455.625,E2 -14455.625} C_VEL
LIN {X 0,Y 336.545,Z 309.031,A -85,B 0,C 180,E1 -14458.535,E2 -14458.535} C_VEL
LIN {X 0,Y 338.709,Z 318.214,A -85,B 0,C 180,E1 -14461.027,E2 -14461.027} C_VEL
LIN {X 0,Y 339.848,Z 325.182,A -85,B 0,C 180,E1 -14462.778,E2 -14462.778} C_VEL
LIN {X 0,Y 339.185,Z 330.74,A -85,B 0,C 180,E1 -14463.995,E2 -14463.995} C_VEL
LIN {X 0,Y 343.034,Z 349.153,A -85,B 0,C 180,E1 -14465.011,E2 -14465.011} C_VEL
LIN {X 0,Y 345.694,Z 366.377,A -85,B 0,C 180,E1 -14465.814,E2 -14465.814} C_VEL
LIN {X 0,Y 346.787,Z 377.998,A -85,B 0,C 180,E1 -14466.279,E2 -14466.279} C_VEL
LIN {X 0,Y 344.271,Z 443.478,A -85,B 0,C 180,E1 -14468.013,E2 -14468.013} C_VEL
LIN {X 0,Y 343.139,Z 457.371,A -85,B 0,C 180,E1 -14468.607,E2 -14468.607} C_VEL
LIN {X 0,Y 341.802,Z 469.874,A -85,B 0,C 180,E1 -14469.387,E2 -14469.387} C_VEL
LIN {X 0,Y 340.326,Z 482.022,A -85,B 0,C 180,E1 -14470.397,E2 -14470.397} C_VEL
LIN {X 0,Y 338.783,Z 493.068,A -85,B 0,C 180,E1 -14471.561,E2 -14471.561} C_VEL
LIN {X 0,Y 337.134,Z 504.109,A -85,B 0,C 180,E1 -14473.035,E2 -14473.035} C_VEL
LIN {X 0,Y 335.7,Z 513.885,A -85,B 0,C 180,E1 -14474.66,E2 -14474.66} C_VEL
LIN {X 0,Y 334.557,Z 522.063,A -85,B 0,C 180,E1 -14476.334,E2 -14476.334} C_VEL
LIN {X 0,Y 333.422,Z 529.228,A -85,B 0,C 180,E1 -14478.144,E2 -14478.144} C_VEL
LIN {X 0,Y 332.666,Z 535.864,A -85,B 0,C 180,E1 -14480.273,E2 -14480.273} C_VEL
LIN {X 0,Y 332.262,Z 540.235,A -85,B 0,C 180,E1 -14482.1,E2 -14482.1} C_VEL
LIN {X 0,Y 332.075,Z 543.8,A -85,B 0,C 180,E1 -14484.105,E2 -14484.105} C_VEL
LIN {X 0,Y 332.048,Z 546.344,A -85,B 0,C 180,E1 -14486.362,E2 -14486.362} C_VEL
LIN {X 0,Y 332.191,Z 547.484,A -85,B 0,C 180,E1 -14488.79,E2 -14488.79} C_VEL
LIN {X 0,Y 332.273,Z 547.408,A -85,B 0,C 180,E1 -14490.002,E2 -14490.002} C_VEL
LIN {X 0,Y 332.26,Z 546.876,A -85,B 0,C 180,E1 -14491.214,E2 -14491.214} C_VEL
LIN {X 0,Y 332.123,Z 545.92,A -85,B 0,C 180,E1 -14492.427,E2 -14492.427} C_VEL
LIN {X 0,Y 332.091,Z 544.545,A -85,B 0,C 180,E1 -14493.642,E2 -14493.642} C_VEL
LIN {X 0,Y 332.114,Z 541.407,A -85,B 0,C 180,E1 -14495.555,E2 -14495.555} C_VEL
LIN {X 0,Y 332.26,Z 537.504,A -85,B 0,C 180,E1 -14497.292,E2 -14497.292} C_VEL
LIN {X 0,Y 332.506,Z 531.147,A -85,B 0,C 180,E1 -14499.429,E2 -14499.429} C_VEL
LIN {X 0,Y 333.004,Z 524.186,A -85,B 0,C 180,E1 -14501.258,E2 -14501.258} C_VEL
LIN {X 0,Y 333.696,Z 517.075,A -85,B 0,C 180,E1 -14502.777,E2 -14502.777} C_VEL
LIN {X 0,Y 334.525,Z 508.487,A -85,B 0,C 180,E1 -14504.292,E2 -14504.292} C_VEL
LIN {X 0,Y 335.308,Z 499.132,A -85,B 0,C 180,E1 -14505.643,E2 -14505.643} C_VEL
LIN {X 0,Y 336.47,Z 487.365,A -85,B 0,C 180,E1 -14507.003,E2 -14507.003} C_VEL
LIN {X 0,Y 337.396,Z 475.91,A -85,B 0,C 180,E1 -14508.05,E2 -14508.05} C_VEL
LIN {X 0,Y 338.428,Z 463.004,A -85,B 0,C 180,E1 -14508.934,E2 -14508.934} C_VEL
LIN {X 0,Y 339.233,Z 449.514,A -85,B 0,C 180,E1 -14509.594,E2 -14509.594} C_VEL
LIN {X 0,Y 339.718,Z 434.666,A -85,B 0,C 180,E1 -14510.038,E2 -14510.038} C_VEL
LIN {X 0,Y 341.11,Z 374.773,A -85,B 0,C 180,E1 -14511.517,E2 -14511.517} C_VEL
LIN {X 0,Y 336.222,Z 335.657,A -85,B 0,C 180,E1 -14512.815,E2 -14512.815} C_VEL
LIN {X 0,Y 337.831,Z 320.971,A -85,B 0,C 180,E1 -14516.22,E2 -14516.22} C_VEL
LIN {X 0,Y 337.068,Z 315.253,A -85,B 0,C 180,E1 -14517.64,E2 -14517.64} C_VEL
LIN {X 0,Y 334.689,Z 303.86,A -85,B 0,C 180,E1 -14520.576,E2 -14520.576} C_VEL
LIN {X 0,Y 333.681,Z 298.922,A -85,B 0,C 180,E1 -14521.911,E2 -14521.911} C_VEL
LIN {X 0,Y 333.68,Z 298.923,A -85,B 0,C 180,E1 -14524.772,E2 -14524.772} C_VEL
LIN {X 0,Y 333.637,Z 298.922,A -85,B 0,C 180,E1 -14527.651,E2 -14527.651} C_VEL
LIN {X 0,Y 333.596,Z 298.933,A -85,B 0,C 180,E1 -14530.772,E2 -14530.772} C_VEL
LIN {X 0,Y 333.58,Z 298.93,A -85,B 0,C 180,E1 -14534.247,E2 -14534.247} C_VEL
LIN {X 0,Y 333.611,Z 298.926,A -85,B 0,C 180,E1 -14537.613,E2 -14537.613} C_VEL
LIN {X 0,Y 333.603,Z 298.93,A -85,B 0,C 180,E1 -14541.208,E2 -14541.208} C_VEL
LIN {X 0,Y 333.659,Z 298.92,A -85,B 0,C 180,E1 -14543.858,E2 -14543.858} C_VEL
LIN {X 0,Y 333.622,Z 298.927,A -85,B 0,C 180,E1 -14547.413,E2 -14547.413} C_VEL
LIN {X 0,Y 333.65,Z 298.926,A -85,B 0,C 180,E1 -14551.021,E2 -14551.021} C_VEL
LIN {X 0,Y 333.679,Z 298.923,A -85,B 0,C 180,E1 -14555.086,E2 -14555.086} C_VEL
LIN {X 0,Y 333.635,Z 298.927,A -85,B 0,C 180,E1 -14559.016,E2 -14559.016} C_VEL
LIN {X 0,Y 333.719,Z 298.915,A -85,B 0,C 180,E1 -14561.585,E2 -14561.585} C_VEL
LIN {X 0,Y 333.788,Z 298.907,A -85,B 0,C 180,E1 -14565.576,E2 -14565.576} C_VEL
LIN {X 0,Y 333.794,Z 298.907,A -85,B 0,C 180,E1 -14569.076,E2 -14569.076} C_VEL
LIN {X 0,Y 333.98,Z 298.881,A -85,B 0,C 180,E1 -14572.746,E2 -14572.746} C_VEL
LIN {X 0,Y 333.775,Z 298.909,A -85,B 0,C 180,E1 -14575.168,E2 -14575.168} C_VEL
LIN {X 0,Y 334.075,Z 298.873,A -85,B 0,C 180,E1 -14577.588,E2 -14577.588} C_VEL
LIN {X 0,Y 334.164,Z 298.858,A -85,B 0,C 180,E1 -14579.999,E2 -14579.999} C_VEL
LIN {X 0,Y 334.075,Z 298.868,A -85,B 0,C 180,E1 -14582.411,E2 -14582.411} C_VEL
LIN {X 0,Y 333.963,Z 298.882,A -85,B 0,C 180,E1 -14586.721,E2 -14586.721} C_VEL
LIN {X 0,Y 333.827,Z 298.904,A -85,B 0,C 180,E1 -14589.695,E2 -14589.695} C_VEL
LIN {X 0,Y 333.77,Z 298.91,A -85,B 0,C 180,E1 -14593.392,E2 -14593.392} C_VEL
LIN {X 0,Y 333.732,Z 298.915,A -85,B 0,C 180,E1 -14595.888,E2 -14595.888} C_VEL
LIN {X 0,Y 333.636,Z 298.928,A -85,B 0,C 180,E1 -14599.696,E2 -14599.696} C_VEL
LIN {X 0,Y 333.648,Z 298.925,A -85,B 0,C 180,E1 -14603.591,E2 -14603.591} C_VEL
LIN {X 0,Y 333.714,Z 298.915,A -85,B 0,C 180,E1 -14606.247,E2 -14606.247} C_VEL
LIN {X 0,Y 333.691,Z 298.916,A -85,B 0,C 180,E1 -14608.973,E2 -14608.973} C_VEL
LIN {X 0,Y 333.625,Z 298.925,A -85,B 0,C 180,E1 -14612.588,E2 -14612.588} C_VEL
LIN {X 0,Y 333.659,Z 298.924,A -85,B 0,C 180,E1 -14616.14,E2 -14616.14} C_VEL
LIN {X 0,Y 333.637,Z 298.923,A -85,B 0,C 180,E1 -14619.193,E2 -14619.193} C_VEL
LIN {X 0,Y 333.624,Z 298.926,A -85,B 0,C 180,E1 -14622.502,E2 -14622.502} C_VEL
LIN {X 0,Y 333.647,Z 298.927,A -85,B 0,C 180,E1 -14625.966,E2 -14625.966} C_VEL
LIN {X 0,Y 333.691,Z 298.916,A -85,B 0,C 180,E1 -14629.306,E2 -14629.306} C_VEL
LIN {X 0,Y 333.658,Z 298.92,A -85,B 0,C 180,E1 -14633.168,E2 -14633.168} C_VEL
LIN {X 0,Y 333.629,Z 298.925,A -85,B 0,C 180,E1 -14636.792,E2 -14636.792} C_VEL
LIN {X 0,Y 333.688,Z 298.918,A -85,B 0,C 180,E1 -14639.713,E2 -14639.713} C_VEL
LIN {X 0,Y 333.734,Z 298.915,A -85,B 0,C 180,E1 -14642.401,E2 -14642.401} C_VEL
LIN {X 0,Y 333.722,Z 298.912,A -85,B 0,C 180,E1 -14645.091,E2 -14645.091} C_VEL
LIN {X 0,Y 333.678,Z 298.918,A -85,B 0,C 180,E1 -14649.019,E2 -14649.019} C_VEL
LIN {X 0,Y 333.791,Z 298.903,A -85,B 0,C 180,E1 -14651.589,E2 -14651.589} C_VEL
LIN {X 0,Y 333.806,Z 298.902,A -85,B 0,C 180,E1 -14655.576,E2 -14655.576} C_VEL
LIN {X 0,Y 333.831,Z 298.899,A -85,B 0,C 180,E1 -14659.077,E2 -14659.077} C_VEL
LIN {X 0,Y 334.023,Z 298.878,A -85,B 0,C 180,E1 -14662.746,E2 -14662.746} C_VEL
LIN {X 0,Y 333.807,Z 298.902,A -85,B 0,C 180,E1 -14665.168,E2 -14665.168} C_VEL
LIN {X 0,Y 334.104,Z 298.864,A -85,B 0,C 180,E1 -14667.587,E2 -14667.587} C_VEL
LIN {X 0,Y 334.245,Z 298.848,A -85,B 0,C 180,E1 -14669.998,E2 -14669.998} C_VEL
LIN {X 0,Y 334.104,Z 298.868,A -85,B 0,C 180,E1 -14672.409,E2 -14672.409} C_VEL
LIN {X 0,Y 334.018,Z 298.876,A -85,B 0,C 180,E1 -14677.25,E2 -14677.25} C_VEL
LIN {X 0,Y 333.83,Z 298.903,A -85,B 0,C 180,E1 -14680.919,E2 -14680.919} C_VEL
LIN {X 0,Y 333.8,Z 298.906,A -85,B 0,C 180,E1 -14684.631,E2 -14684.631} C_VEL
LIN {X 0,Y 333.788,Z 298.907,A -85,B 0,C 180,E1 -14688.653,E2 -14688.653} C_VEL
LIN {X 0,Y 333.682,Z 298.917,A -85,B 0,C 180,E1 -14692.274,E2 -14692.274} C_VEL
LIN {X 0,Y 333.722,Z 298.912,A -85,B 0,C 180,E1 -14696.242,E2 -14696.242} C_VEL
LIN {X 0,Y 333.695,Z 298.921,A -85,B 0,C 180,E1 -14698.968,E2 -14698.968} C_VEL
LIN {X 0,Y 333.624,Z 298.925,A -85,B 0,C 180,E1 -14702.583,E2 -14702.583} C_VEL
LIN {X 0,Y 333.655,Z 298.92,A -85,B 0,C 180,E1 -14706.135,E2 -14706.135} C_VEL
LIN {X 0,Y 333.738,Z 299.103,A -85,B 0,C 180,E1 -14709.113,E2 -14709.113} C_VEL
LIN {X 0,Y 334.567,Z 301.601,A -85,B 0,C 180,E1 -14709.27,E2 -14709.27} C_VEL
LIN {X 0,Y 341.874,Z 324.198,A -85,B 0,C 180,E1 -14710.273,E2 -14710.273} C_VEL
LIN {X 0,Y 339.779,Z 407.312,A -85,B 0,C 180,E1 -14712.345,E2 -14712.345} C_VEL
LIN {X 0,Y 339.291,Z 420.584,A -85,B 0,C 180,E1 -14712.909,E2 -14712.909} C_VEL
LIN {X 0,Y 338.547,Z 433.846,A -85,B 0,C 180,E1 -14713.725,E2 -14713.725} C_VEL
LIN {X 0,Y 337.699,Z 446.151,A -85,B 0,C 180,E1 -14714.751,E2 -14714.751} C_VEL
LIN {X 0,Y 336.822,Z 456.699,A -85,B 0,C 180,E1 -14715.863,E2 -14715.863} C_VEL
LIN {X 0,Y 335.897,Z 467.414,A -85,B 0,C 180,E1 -14717.272,E2 -14717.272} C_VEL
LIN {X 0,Y 335.792,Z 468.482,A -85,B 0,C 180,E1 -14717.433,E2 -14717.433} C_VEL
LIN {X 0,Y 334.707,Z 472.858,A -85,B 0,C 180,E1 -14718.094,E2 -14718.094} C_VEL
LIN {X 0,Y 331.182,Z 479.578,A -85,B 0,C 180,E1 -14719.198,E2 -14719.198} C_VEL
LIN {X 0,Y 327.712,Z 485.758,A -85,B 0,C 180,E1 -14720.407,E2 -14720.407} C_VEL
LIN {X 0,Y 326.725,Z 489.222,A -85,B 0,C 180,E1 -14721.223,E2 -14721.223} C_VEL
LIN {X 0,Y 326.172,Z 495.238,A -85,B 0,C 180,E1 -14722.893,E2 -14722.893} C_VEL
LIN {X 0,Y 325.63,Z 501.411,A -85,B 0,C 180,E1 -14725.087,E2 -14725.087} C_VEL
LIN {X 0,Y 325.263,Z 506.026,A -85,B 0,C 180,E1 -14727.305,E2 -14727.305} C_VEL
LIN {X 0,Y 325.03,Z 508.187,A -85,B 0,C 180,E1 -14728.739,E2 -14728.739} C_VEL
LIN {X 0,Y 324.907,Z 509.776,A -85,B 0,C 180,E1 -14730.166,E2 -14730.166} C_VEL
LIN {X 0,Y 324.928,Z 511.129,A -85,B 0,C 180,E1 -14732.459,E2 -14732.459} C_VEL
LIN {X 0,Y 325.047,Z 511.177,A -85,B 0,C 180,E1 -14734.379,E2 -14734.379} C_VEL
LIN {X 0,Y 325.262,Z 510.573,A -85,B 0,C 180,E1 -14735.762,E2 -14735.762} C_VEL
LIN {X 0,Y 325.774,Z 508.472,A -85,B 0,C 180,E1 -14738.051,E2 -14738.051} C_VEL
LIN {X 0,Y 326.328,Z 505.756,A -85,B 0,C 180,E1 -14739.844,E2 -14739.844} C_VEL
LIN {X 0,Y 327.09,Z 501.592,A -85,B 0,C 180,E1 -14741.848,E2 -14741.848} C_VEL
LIN {X 0,Y 328.155,Z 496.055,A -85,B 0,C 180,E1 -14743.835,E2 -14743.835} C_VEL
LIN {X 0,Y 329.494,Z 489.01,A -85,B 0,C 180,E1 -14745.802,E2 -14745.802} C_VEL
LIN {X 0,Y 330.943,Z 480.827,A -85,B 0,C 180,E1 -14747.617,E2 -14747.617} C_VEL
LIN {X 0,Y 332.384,Z 472.001,A -85,B 0,C 180,E1 -14749.185,E2 -14749.185} C_VEL
LIN {X 0,Y 333.899,Z 462.59,A -85,B 0,C 180,E1 -14750.538,E2 -14750.538} C_VEL
LIN {X 0,Y 335.4,Z 451.243,A -85,B 0,C 180,E1 -14751.869,E2 -14751.869} C_VEL
LIN {X 0,Y 336.733,Z 439.299,A -85,B 0,C 180,E1 -14752.957,E2 -14752.957} C_VEL
LIN {X 0,Y 337.846,Z 427.083,A -85,B 0,C 180,E1 -14753.806,E2 -14753.806} C_VEL
LIN {X 0,Y 338.645,Z 414.455,A -85,B 0,C 180,E1 -14754.442,E2 -14754.442} C_VEL
LIN {X 0,Y 339.423,Z 397.036,A -85,B 0,C 180,E1 -14754.974,E2 -14754.974} C_VEL
LIN {X 0,Y 342.153,Z 331.281,A -85,B 0,C 180,E1 -14756.746,E2 -14756.746} C_VEL
LIN {X 0,Y 338.156,Z 322.206,A -85,B 0,C 180,E1 -14757.501,E2 -14757.501} C_VEL
LIN {X 0,Y 331.141,Z 308.394,A -85,B 0,C 180,E1 -14758.829,E2 -14758.829} C_VEL
LIN {X 0,Y 327.873,Z 302.35,A -85,B 0,C 180,E1 -14759.496,E2 -14759.496} C_VEL
LIN {X 0,Y 327.09,Z 299.743,A -85,B 0,C 180,E1 -14760.308,E2 -14760.308} C_VEL
LIN {X 0,Y 327,Z 299.753,A -85,B 0,C 180,E1 -14762.464,E2 -14762.464} C_VEL
LIN {X 0,Y 326.941,Z 299.759,A -85,B 0,C 180,E1 -14766.171,E2 -14766.171} C_VEL
LIN {X 0,Y 326.762,Z 299.781,A -85,B 0,C 180,E1 -14769.908,E2 -14769.908} C_VEL
LIN {X 0,Y 326.714,Z 299.789,A -85,B 0,C 180,E1 -14773.688,E2 -14773.688} C_VEL
LIN {X 0,Y 326.62,Z 299.794,A -85,B 0,C 180,E1 -14777.533,E2 -14777.533} C_VEL
LIN {X 0,Y 326.571,Z 299.806,A -85,B 0,C 180,E1 -14781.461,E2 -14781.461} C_VEL
LIN {X 0,Y 326.635,Z 299.792,A -85,B 0,C 180,E1 -14785.489,E2 -14785.489} C_VEL
LIN {X 0,Y 326.609,Z 299.799,A -85,B 0,C 180,E1 -14788.256,E2 -14788.256} C_VEL
LIN {X 0,Y 326.538,Z 299.807,A -85,B 0,C 180,E1 -14791.102,E2 -14791.102} C_VEL
LIN {X 0,Y 326.574,Z 299.801,A -85,B 0,C 180,E1 -14794.024,E2 -14794.024} C_VEL
LIN {X 0,Y 326.598,Z 299.798,A -85,B 0,C 180,E1 -14797.243,E2 -14797.243} C_VEL
LIN {X 0,Y 326.575,Z 299.802,A -85,B 0,C 180,E1 -14800.212,E2 -14800.212} C_VEL
LIN {X 0,Y 326.538,Z 299.811,A -85,B 0,C 180,E1 -14803.53,E2 -14803.53} C_VEL
LIN {X 0,Y 326.553,Z 299.807,A -85,B 0,C 180,E1 -14807.033,E2 -14807.033} C_VEL
LIN {X 0,Y 326.592,Z 299.802,A -85,B 0,C 180,E1 -14810.778,E2 -14810.778} C_VEL
LIN {X 0,Y 326.596,Z 299.808,A -85,B 0,C 180,E1 -14814.485,E2 -14814.485} C_VEL
LIN {X 0,Y 326.639,Z 300.03,A -85,B 0,C 180,E1 -14814.793,E2 -14814.793} C_VEL
LIN {X 0,Y 329.808,Z 310.737,A -85,B 0,C 180,E1 -14818.094,E2 -14818.094} C_VEL
LIN {X 0,Y 332.128,Z 320.742,A -85,B 0,C 180,E1 -14820.882,E2 -14820.882} C_VEL
LIN {X 0,Y 333.143,Z 326.466,A -85,B 0,C 180,E1 -14822.38,E2 -14822.38} C_VEL
LIN {X 0,Y 332.795,Z 330.337,A -85,B 0,C 180,E1 -14823.233,E2 -14823.233} C_VEL
LIN {X 0,Y 337.01,Z 350.307,A -85,B 0,C 180,E1 -14824.392,E2 -14824.392} C_VEL
LIN {X 0,Y 339.655,Z 367.868,A -85,B 0,C 180,E1 -14825.246,E2 -14825.246} C_VEL
LIN {X 0,Y 340.681,Z 378.172,A -85,B 0,C 180,E1 -14825.676,E2 -14825.676} C_VEL
LIN {X 0,Y 338.059,Z 442.63,A -85,B 0,C 180,E1 -14827.426,E2 -14827.426} C_VEL
LIN {X 0,Y 336.887,Z 456.511,A -85,B 0,C 180,E1 -14828.029,E2 -14828.029} C_VEL
LIN {X 0,Y 335.445,Z 469.065,A -85,B 0,C 180,E1 -14828.818,E2 -14828.818} C_VEL
LIN {X 0,Y 333.894,Z 481.262,A -85,B 0,C 180,E1 -14829.842,E2 -14829.842} C_VEL
LIN {X 0,Y 332.247,Z 492.379,A -85,B 0,C 180,E1 -14831.025,E2 -14831.025} C_VEL
LIN {X 0,Y 330.705,Z 502.482,A -85,B 0,C 180,E1 -14832.376,E2 -14832.376} C_VEL
LIN {X 0,Y 329.231,Z 511.718,A -85,B 0,C 180,E1 -14833.892,E2 -14833.892} C_VEL
LIN {X 0,Y 328.096,Z 519.397,A -85,B 0,C 180,E1 -14835.426,E2 -14835.426} C_VEL
LIN {X 0,Y 326.838,Z 526.995,A -85,B 0,C 180,E1 -14837.27,E2 -14837.27} C_VEL
LIN {X 0,Y 326.001,Z 532.185,A -85,B 0,C 180,E1 -14838.815,E2 -14838.815} C_VEL
LIN {X 0,Y 325.464,Z 537.276,A -85,B 0,C 180,E1 -14840.683,E2 -14840.683} C_VEL
LIN {X 0,Y 325.111,Z 541.214,A -85,B 0,C 180,E1 -14842.55,E2 -14842.55} C_VEL
LIN {X 0,Y 324.999,Z 543.721,A -85,B 0,C 180,E1 -14844.122,E2 -14844.122} C_VEL
LIN {X 0,Y 324.971,Z 546.008,A -85,B 0,C 180,E1 -14846.282,E2 -14846.282} C_VEL
LIN {X 0,Y 324.957,Z 546.748,A -85,B 0,C 180,E1 -14847.523,E2 -14847.523} C_VEL
LIN {X 0,Y 325.093,Z 547.085,A -85,B 0,C 180,E1 -14848.763,E2 -14848.763} C_VEL
LIN {X 0,Y 325.214,Z 546.957,A -85,B 0,C 180,E1 -14850.002,E2 -14850.002} C_VEL
LIN {X 0,Y 325.18,Z 546.397,A -85,B 0,C 180,E1 -14851.24,E2 -14851.24} C_VEL
LIN {X 0,Y 325.031,Z 545.413,A -85,B 0,C 180,E1 -14852.48,E2 -14852.48} C_VEL
LIN {X 0,Y 325.019,Z 543.991,A -85,B 0,C 180,E1 -14853.721,E2 -14853.721} C_VEL
LIN {X 0,Y 325.025,Z 541.118,A -85,B 0,C 180,E1 -14855.504,E2 -14855.504} C_VEL
LIN {X 0,Y 325.182,Z 536.807,A -85,B 0,C 180,E1 -14857.452,E2 -14857.452} C_VEL
LIN {X 0,Y 325.462,Z 530.358,A -85,B 0,C 180,E1 -14859.635,E2 -14859.635} C_VEL
LIN {X 0,Y 326.001,Z 523.307,A -85,B 0,C 180,E1 -14861.504,E2 -14861.504} C_VEL
LIN {X 0,Y 326.701,Z 516.088,A -85,B 0,C 180,E1 -14863.055,E2 -14863.055} C_VEL
LIN {X 0,Y 327.65,Z 506.331,A -85,B 0,C 180,E1 -14864.757,E2 -14864.757} C_VEL
LIN {X 0,Y 328.581,Z 496.52,A -85,B 0,C 180,E1 -14866.145,E2 -14866.145} C_VEL
LIN {X 0,Y 329.575,Z 485.831,A -85,B 0,C 180,E1 -14867.37,E2 -14867.37} C_VEL
LIN {X 0,Y 330.633,Z 473.994,A -85,B 0,C 180,E1 -14868.433,E2 -14868.433} C_VEL
LIN {X 0,Y 331.655,Z 460.632,A -85,B 0,C 180,E1 -14869.336,E2 -14869.336} C_VEL
LIN {X 0,Y 332.426,Z 448.001,A -85,B 0,C 180,E1 -14869.932,E2 -14869.932} C_VEL
LIN {X 0,Y 332.88,Z 432.581,A -85,B 0,C 180,E1 -14870.387,E2 -14870.387} C_VEL
LIN {X 0,Y 334.275,Z 375.39,A -85,B 0,C 180,E1 -14871.838,E2 -14871.838} C_VEL
LIN {X 0,Y 329.34,Z 335.295,A -85,B 0,C 180,E1 -14873.204,E2 -14873.204} C_VEL
LIN {X 0,Y 330.834,Z 321.414,A -85,B 0,C 180,E1 -14876.494,E2 -14876.494} C_VEL
LIN {X 0,Y 329.206,Z 311.961,A -85,B 0,C 180,E1 -14878.921,E2 -14878.921} C_VEL
LIN {X 0,Y 326.629,Z 299.8,A -85,B 0,C 180,E1 -14882.221,E2 -14882.221} C_VEL
LIN {X 0,Y 326.606,Z 299.798,A -85,B 0,C 180,E1 -14885.519,E2 -14885.519} C_VEL
LIN {X 0,Y 326.567,Z 299.805,A -85,B 0,C 180,E1 -14889.217,E2 -14889.217} C_VEL
LIN {X 0,Y 326.563,Z 299.808,A -85,B 0,C 180,E1 -14892.969,E2 -14892.969} C_VEL
LIN {X 0,Y 326.553,Z 299.809,A -85,B 0,C 180,E1 -14897.029,E2 -14897.029} C_VEL
LIN {X 0,Y 326.574,Z 299.806,A -85,B 0,C 180,E1 -14900.777,E2 -14900.777} C_VEL
LIN {X 0,Y 326.596,Z 299.801,A -85,B 0,C 180,E1 -14904.478,E2 -14904.478} C_VEL
LIN {X 0,Y 326.587,Z 299.803,A -85,B 0,C 180,E1 -14907.453,E2 -14907.453} C_VEL
LIN {X 0,Y 326.605,Z 299.799,A -85,B 0,C 180,E1 -14910.335,E2 -14910.335} C_VEL
LIN {X 0,Y 326.602,Z 299.805,A -85,B 0,C 180,E1 -14913.134,E2 -14913.134} C_VEL
LIN {X 0,Y 326.611,Z 299.798,A -85,B 0,C 180,E1 -14915.867,E2 -14915.867} C_VEL
LIN {X 0,Y 326.592,Z 299.801,A -85,B 0,C 180,E1 -14919.86,E2 -14919.86} C_VEL
LIN {X 0,Y 326.686,Z 299.79,A -85,B 0,C 180,E1 -14923.759,E2 -14923.759} C_VEL
LIN {X 0,Y 326.735,Z 299.782,A -85,B 0,C 180,E1 -14926.313,E2 -14926.313} C_VEL
LIN {X 0,Y 326.762,Z 299.779,A -85,B 0,C 180,E1 -14930.092,E2 -14930.092} C_VEL
LIN {X 0,Y 326.931,Z 299.758,A -85,B 0,C 180,E1 -14932.589,E2 -14932.589} C_VEL
LIN {X 0,Y 326.961,Z 299.756,A -85,B 0,C 180,E1 -14933.83,E2 -14933.83} C_VEL
LIN {X 0,Y 327.016,Z 299.752,A -85,B 0,C 180,E1 -14937.536,E2 -14937.536} C_VEL
LIN {X 0,Y 327.117,Z 299.736,A -85,B 0,C 180,E1 -14939.999,E2 -14939.999} C_VEL
LIN {X 0,Y 327.016,Z 299.747,A -85,B 0,C 180,E1 -14942.463,E2 -14942.463} C_VEL
LIN {X 0,Y 326.917,Z 299.76,A -85,B 0,C 180,E1 -14946.718,E2 -14946.718} C_VEL
LIN {X 0,Y 326.783,Z 299.779,A -85,B 0,C 180,E1 -14949.907,E2 -14949.907} C_VEL
LIN {X 0,Y 326.734,Z 299.788,A -85,B 0,C 180,E1 -14953.686,E2 -14953.686} C_VEL
LIN {X 0,Y 326.63,Z 299.8,A -85,B 0,C 180,E1 -14957.531,E2 -14957.531} C_VEL
LIN {X 0,Y 326.588,Z 299.804,A -85,B 0,C 180,E1 -14961.458,E2 -14961.458} C_VEL
LIN {X 0,Y 326.67,Z 299.793,A -85,B 0,C 180,E1 -14965.485,E2 -14965.485} C_VEL
LIN {X 0,Y 326.642,Z 299.798,A -85,B 0,C 180,E1 -14969.66,E2 -14969.66} C_VEL
LIN {X 0,Y 326.589,Z 299.805,A -85,B 0,C 180,E1 -14974.021,E2 -14974.021} C_VEL
LIN {X 0,Y 326.612,Z 299.798,A -85,B 0,C 180,E1 -14977.239,E2 -14977.239} C_VEL
LIN {X 0,Y 326.57,Z 299.803,A -85,B 0,C 180,E1 -14981.133,E2 -14981.133} C_VEL
LIN {X 0,Y 326.558,Z 299.805,A -85,B 0,C 180,E1 -14984.751,E2 -14984.751} C_VEL
LIN {X 0,Y 326.611,Z 299.803,A -85,B 0,C 180,E1 -14988.162,E2 -14988.162} C_VEL
LIN {X 0,Y 326.636,Z 299.795,A -85,B 0,C 180,E1 -14991.395,E2 -14991.395} C_VEL
LIN {X 0,Y 326.611,Z 299.798,A -85,B 0,C 180,E1 -14994.852,E2 -14994.852} C_VEL
LIN {X 0,Y 326.6,Z 299.799,A -85,B 0,C 180,E1 -14997.456,E2 -14997.456} C_VEL
LIN {X 0,Y 326.641,Z 299.799,A -85,B 0,C 180,E1 -15000.34,E2 -15000.34} C_VEL
LIN {X 0,Y 326.685,Z 299.792,A -85,B 0,C 180,E1 -15004.516,E2 -15004.516} C_VEL
LIN {X 0,Y 326.643,Z 299.798,A -85,B 0,C 180,E1 -15008.545,E2 -15008.545} C_VEL
LIN {X 0,Y 326.742,Z 299.782,A -85,B 0,C 180,E1 -15011.177,E2 -15011.177} C_VEL
LIN {X 0,Y 326.761,Z 299.779,A -85,B 0,C 180,E1 -15015.432,E2 -15015.432} C_VEL
LIN {X 0,Y 326.768,Z 299.781,A -85,B 0,C 180,E1 -15018.838,E2 -15018.838} C_VEL
LIN {X 0,Y 326.977,Z 299.758,A -85,B 0,C 180,E1 -15022.589,E2 -15022.589} C_VEL
LIN {X 0,Y 326.775,Z 299.779,A -85,B 0,C 180,E1 -15025.063,E2 -15025.063} C_VEL
LIN {X 0,Y 327.045,Z 299.743,A -85,B 0,C 180,E1 -15027.535,E2 -15027.535} C_VEL
LIN {X 0,Y 327.196,Z 299.725,A -85,B 0,C 180,E1 -15029.998,E2 -15029.998} C_VEL
LIN {X 0,Y 327.045,Z 299.747,A -85,B 0,C 180,E1 -15032.461,E2 -15032.461} C_VEL
LIN {X 0,Y 326.99,Z 299.751,A -85,B 0,C 180,E1 -15036.167,E2 -15036.167} C_VEL
LIN {X 0,Y 326.909,Z 299.765,A -85,B 0,C 180,E1 -15038.652,E2 -15038.652} C_VEL
LIN {X 0,Y 326.731,Z 299.785,A -85,B 0,C 180,E1 -15042.418,E2 -15042.418} C_VEL
LIN {X 0,Y 326.746,Z 299.786,A -85,B 0,C 180,E1 -15044.954,E2 -15044.954} C_VEL
LIN {X 0,Y 326.754,Z 299.785,A -85,B 0,C 180,E1 -15048.851,E2 -15048.851} C_VEL
LIN {X 0,Y 326.612,Z 299.802,A -85,B 0,C 180,E1 -15052.783,E2 -15052.783} C_VEL
LIN {X 0,Y 326.678,Z 299.791,A -85,B 0,C 180,E1 -15055.48,E2 -15055.48} C_VEL
LIN {X 0,Y 326.644,Z 299.794,A -85,B 0,C 180,E1 -15059.655,E2 -15059.655} C_VEL
LIN {X 0,Y 326.587,Z 299.8,A -85,B 0,C 180,E1 -15064.016,E2 -15064.016} C_VEL
LIN {X 0,Y 326.609,Z 299.803,A -85,B 0,C 180,E1 -15067.235,E2 -15067.235} C_VEL
LIN {X 0,Y 326.653,Z 299.796,A -85,B 0,C 180,E1 -15068.769,E2 -15068.769} C_VEL
LIN {X 0,Y 335.151,Z 325.493,A -85,B 0,C 180,E1 -15069.948,E2 -15069.948} C_VEL
LIN {X 0,Y 332.902,Z 407.928,A -85,B 0,C 180,E1 -15072.054,E2 -15072.054} C_VEL
LIN {X 0,Y 332.403,Z 421.246,A -85,B 0,C 180,E1 -15072.638,E2 -15072.638} C_VEL
LIN {X 0,Y 331.645,Z 434.335,A -85,B 0,C 180,E1 -15073.465,E2 -15073.465} C_VEL
LIN {X 0,Y 330.763,Z 446.622,A -85,B 0,C 180,E1 -15074.513,E2 -15074.513} C_VEL
LIN {X 0,Y 329.824,Z 457.372,A -85,B 0,C 180,E1 -15075.674,E2 -15075.674} C_VEL
LIN {X 0,Y 328.924,Z 467.769,A -85,B 0,C 180,E1 -15077.074,E2 -15077.074} C_VEL
LIN {X 0,Y 327.978,Z 476.868,A -85,B 0,C 180,E1 -15078.58,E2 -15078.58} C_VEL
LIN {X 0,Y 327.119,Z 485.565,A -85,B 0,C 180,E1 -15080.347,E2 -15080.347} C_VEL
LIN {X 0,Y 326.725,Z 489.222,A -85,B 0,C 180,E1 -15081.223,E2 -15081.223} C_VEL
LIN {X 0,Y 325.778,Z 492.514,A -85,B 0,C 180,E1 -15082.069,E2 -15082.069} C_VEL
LIN {X 0,Y 322.505,Z 497.408,A -85,B 0,C 180,E1 -15083.481,E2 -15083.481} C_VEL
LIN {X 0,Y 319.278,Z 501.61,A -85,B 0,C 180,E1 -15084.985,E2 -15084.985} C_VEL
LIN {X 0,Y 318.424,Z 503.819,A -85,B 0,C 180,E1 -15085.962,E2 -15085.962} C_VEL
LIN {X 0,Y 318.046,Z 507.444,A -85,B 0,C 180,E1 -15087.973,E2 -15087.973} C_VEL
LIN {X 0,Y 317.864,Z 509.512,A -85,B 0,C 180,E1 -15089.561,E2 -15089.561} C_VEL
LIN {X 0,Y 317.815,Z 510.685,A -85,B 0,C 180,E1 -15090.89,E2 -15090.89} C_VEL
LIN {X 0,Y 317.84,Z 511.478,A -85,B 0,C 180,E1 -15092.333,E2 -15092.333} C_VEL
LIN {X 0,Y 317.895,Z 511.687,A -85,B 0,C 180,E1 -15093.759,E2 -15093.759} C_VEL
LIN {X 0,Y 318.067,Z 511.4,A -85,B 0,C 180,E1 -15095.177,E2 -15095.177} C_VEL
LIN {X 0,Y 318.353,Z 510.592,A -85,B 0,C 180,E1 -15096.587,E2 -15096.587} C_VEL
LIN {X 0,Y 318.68,Z 509.271,A -85,B 0,C 180,E1 -15097.982,E2 -15097.982} C_VEL
LIN {X 0,Y 319.348,Z 506.35,A -85,B 0,C 180,E1 -15100.056,E2 -15100.056} C_VEL
LIN {X 0,Y 320.153,Z 502.252,A -85,B 0,C 180,E1 -15102.102,E2 -15102.102} C_VEL
LIN {X 0,Y 321.326,Z 496.564,A -85,B 0,C 180,E1 -15104.202,E2 -15104.202} C_VEL
LIN {X 0,Y 322.693,Z 489.795,A -85,B 0,C 180,E1 -15106.139,E2 -15106.139} C_VEL
LIN {X 0,Y 324.202,Z 481.894,A -85,B 0,C 180,E1 -15107.948,E2 -15107.948} C_VEL
LIN {X 0,Y 325.764,Z 473.005,A -85,B 0,C 180,E1 -15109.591,E2 -15109.591} C_VEL
LIN {X 0,Y 327.602,Z 462.186,A -85,B 0,C 180,E1 -15111.178,E2 -15111.178} C_VEL
LIN {X 0,Y 329.145,Z 451.047,A -85,B 0,C 180,E1 -15112.486,E2 -15112.486} C_VEL
LIN {X 0,Y 330.564,Z 438.902,A -85,B 0,C 180,E1 -15113.592,E2 -15113.592} C_VEL
LIN {X 0,Y 331.712,Z 426.63,A -85,B 0,C 180,E1 -15114.443,E2 -15114.443} C_VEL
LIN {X 0,Y 332.516,Z 414.472,A -85,B 0,C 180,E1 -15115.049,E2 -15115.049} C_VEL
LIN {X 0,Y 333.375,Z 395.062,A -85,B 0,C 180,E1 -15115.647,E2 -15115.647} C_VEL
LIN {X 0,Y 336.209,Z 333.358,A -85,B 0,C 180,E1 -15117.353,E2 -15117.353} C_VEL
LIN {X 0,Y 331.802,Z 323.781,A -85,B 0,C 180,E1 -15118.208,E2 -15118.208} C_VEL
LIN {X 0,Y 326.071,Z 312.317,A -85,B 0,C 180,E1 -15119.364,E2 -15119.364} C_VEL
LIN {X 0,Y 320.791,Z 303.033,A -85,B 0,C 180,E1 -15120.471,E2 -15120.471} C_VEL
LIN {X 0,Y 319.979,Z 300.627,A -85,B 0,C 180,E1 -15121.338,E2 -15121.338} C_VEL
LIN {X 0,Y 319.699,Z 300.663,A -85,B 0,C 180,E1 -15125.045,E2 -15125.045} C_VEL
LIN {X 0,Y 319.864,Z 300.642,A -85,B 0,C 180,E1 -15127.576,E2 -15127.576} C_VEL
LIN {X 0,Y 319.68,Z 300.666,A -85,B 0,C 180,E1 -15131.412,E2 -15131.412} C_VEL
LIN {X 0,Y 319.67,Z 300.663,A -85,B 0,C 180,E1 -15134.712,E2 -15134.712} C_VEL
LIN {X 0,Y 319.571,Z 300.672,A -85,B 0,C 180,E1 -15137.933,E2 -15137.933} C_VEL
LIN {X 0,Y 319.526,Z 300.682,A -85,B 0,C 180,E1 -15141.958,E2 -15141.958} C_VEL
LIN {X 0,Y 319.571,Z 300.671,A -85,B 0,C 180,E1 -15146.094,E2 -15146.094} C_VEL
LIN {X 0,Y 319.531,Z 300.678,A -85,B 0,C 180,E1 -15148.94,E2 -15148.94} C_VEL
LIN {X 0,Y 319.49,Z 300.682,A -85,B 0,C 180,E1 -15151.867,E2 -15151.867} C_VEL
LIN {X 0,Y 319.549,Z 300.681,A -85,B 0,C 180,E1 -15155.547,E2 -15155.547} C_VEL
LIN {X 0,Y 319.552,Z 300.679,A -85,B 0,C 180,E1 -15158.012,E2 -15158.012} C_VEL
LIN {X 0,Y 319.505,Z 300.684,A -85,B 0,C 180,E1 -15161.602,E2 -15161.602} C_VEL
LIN {X 0,Y 319.464,Z 300.691,A -85,B 0,C 180,E1 -15165.261,E2 -15165.261} C_VEL
LIN {X 0,Y 319.507,Z 300.684,A -85,B 0,C 180,E1 -15168.716,E2 -15168.716} C_VEL
LIN {X 0,Y 319.543,Z 300.681,A -85,B 0,C 180,E1 -15172.353,E2 -15172.353} C_VEL
LIN {X 0,Y 319.552,Z 300.797,A -85,B 0,C 180,E1 -15173.828,E2 -15173.828} C_VEL
LIN {X 0,Y 322.81,Z 311.569,A -85,B 0,C 180,E1 -15177.335,E2 -15177.335} C_VEL
LIN {X 0,Y 325.164,Z 321.351,A -85,B 0,C 180,E1 -15180.196,E2 -15180.196} C_VEL
LIN {X 0,Y 326.506,Z 329.169,A -85,B 0,C 180,E1 -15182.298,E2 -15182.298} C_VEL
LIN {X 0,Y 326.501,Z 329.773,A -85,B 0,C 180,E1 -15182.415,E2 -15182.415} C_VEL
LIN {X 0,Y 331.054,Z 351.302,A -85,B 0,C 180,E1 -15183.731,E2 -15183.731} C_VEL
LIN {X 0,Y 333.724,Z 369.573,A -85,B 0,C 180,E1 -15184.654,E2 -15184.654} C_VEL
LIN {X 0,Y 334.605,Z 379.351,A -85,B 0,C 180,E1 -15185.077,E2 -15185.077} C_VEL
LIN {X 0,Y 331.87,Z 442.069,A -85,B 0,C 180,E1 -15186.816,E2 -15186.816} C_VEL
LIN {X 0,Y 330.652,Z 455.949,A -85,B 0,C 180,E1 -15187.428,E2 -15187.428} C_VEL
LIN {X 0,Y 329.169,Z 468.524,A -85,B 0,C 180,E1 -15188.229,E2 -15188.229} C_VEL
LIN {X 0,Y 327.487,Z 480.692,A -85,B 0,C 180,E1 -15189.266,E2 -15189.266} C_VEL
LIN {X 0,Y 325.811,Z 491.764,A -85,B 0,C 180,E1 -15190.471,E2 -15190.471} C_VEL
LIN {X 0,Y 323.965,Z 502.847,A -85,B 0,C 180,E1 -15191.997,E2 -15191.997} C_VEL
LIN {X 0,Y 322.367,Z 512.22,A -85,B 0,C 180,E1 -15193.59,E2 -15193.59} C_VEL
LIN {X 0,Y 321.209,Z 519.54,A -85,B 0,C 180,E1 -15195.106,E2 -15195.106} C_VEL
LIN {X 0,Y 319.916,Z 527.049,A -85,B 0,C 180,E1 -15196.99,E2 -15196.99} C_VEL
LIN {X 0,Y 319.001,Z 532.147,A -85,B 0,C 180,E1 -15198.567,E2 -15198.567} C_VEL
LIN {X 0,Y 318.409,Z 537.141,A -85,B 0,C 180,E1 -15200.474,E2 -15200.474} C_VEL
LIN {X 0,Y 318.031,Z 540.999,A -85,B 0,C 180,E1 -15202.383,E2 -15202.383} C_VEL
LIN {X 0,Y 317.904,Z 543.68,A -85,B 0,C 180,E1 -15204.175,E2 -15204.175} C_VEL
LIN {X 0,Y 317.896,Z 545.675,A -85,B 0,C 180,E1 -15206.2,E2 -15206.2} C_VEL
LIN {X 0,Y 317.872,Z 546.386,A -85,B 0,C 180,E1 -15207.468,E2 -15207.468} C_VEL
LIN {X 0,Y 317.998,Z 546.666,A -85,B 0,C 180,E1 -15208.736,E2 -15208.736} C_VEL
LIN {X 0,Y 318.155,Z 546.499,A -85,B 0,C 180,E1 -15210.002,E2 -15210.002} C_VEL
LIN {X 0,Y 318.086,Z 545.904,A -85,B 0,C 180,E1 -15211.268,E2 -15211.268} C_VEL
LIN {X 0,Y 317.942,Z 544.885,A -85,B 0,C 180,E1 -15212.536,E2 -15212.536} C_VEL
LIN {X 0,Y 317.949,Z 543.393,A -85,B 0,C 180,E1 -15213.804,E2 -15213.804} C_VEL
LIN {X 0,Y 318.024,Z 539.647,A -85,B 0,C 180,E1 -15216.033,E2 -15216.033} C_VEL
LIN {X 0,Y 318.159,Z 534.389,A -85,B 0,C 180,E1 -15218.256,E2 -15218.256} C_VEL
LIN {X 0,Y 318.592,Z 527.289,A -85,B 0,C 180,E1 -15220.487,E2 -15220.487} C_VEL
LIN {X 0,Y 319.294,Z 519.57,A -85,B 0,C 180,E1 -15222.393,E2 -15222.393} C_VEL
LIN {X 0,Y 320.056,Z 511.654,A -85,B 0,C 180,E1 -15223.978,E2 -15223.978} C_VEL
LIN {X 0,Y 320.982,Z 501.404,A -85,B 0,C 180,E1 -15225.64,E2 -15225.64} C_VEL
LIN {X 0,Y 322.041,Z 491.226,A -85,B 0,C 180,E1 -15226.971,E2 -15226.971} C_VEL
LIN {X 0,Y 323.036,Z 480.939,A -85,B 0,C 180,E1 -15228.061,E2 -15228.061} C_VEL
LIN {X 0,Y 324.07,Z 468.825,A -85,B 0,C 180,E1 -15229.066,E2 -15229.066} C_VEL
LIN {X 0,Y 325.12,Z 454.994,A -85,B 0,C 180,E1 -15229.905,E2 -15229.905} C_VEL
LIN {X 0,Y 325.814,Z 441.785,A -85,B 0,C 180,E1 -15230.437,E2 -15230.437} C_VEL
LIN {X 0,Y 327.426,Z 375.822,A -85,B 0,C 180,E1 -15232.174,E2 -15232.174} C_VEL
LIN {X 0,Y 322.437,Z 334.872,A -85,B 0,C 180,E1 -15233.61,E2 -15233.61} C_VEL
LIN {X 0,Y 323.82,Z 323.276,A -85,B 0,C 180,E1 -15236.418,E2 -15236.418} C_VEL
LIN {X 0,Y 323.354,Z 319.034,A -85,B 0,C 180,E1 -15237.507,E2 -15237.507} C_VEL
LIN {X 0,Y 320.899,Z 307.062,A -85,B 0,C 180,E1 -15240.715,E2 -15240.715} C_VEL
LIN {X 0,Y 319.565,Z 300.68,A -85,B 0,C 180,E1 -15242.508,E2 -15242.508} C_VEL
LIN {X 0,Y 319.55,Z 300.68,A -85,B 0,C 180,E1 -15246.427,E2 -15246.427} C_VEL
LIN {X 0,Y 319.524,Z 300.68,A -85,B 0,C 180,E1 -15249.66,E2 -15249.66} C_VEL
LIN {X 0,Y 319.51,Z 300.683,A -85,B 0,C 180,E1 -15253.458,E2 -15253.458} C_VEL
LIN {X 0,Y 319.507,Z 300.687,A -85,B 0,C 180,E1 -15257.008,E2 -15257.008} C_VEL
LIN {X 0,Y 319.505,Z 300.684,A -85,B 0,C 180,E1 -15260.364,E2 -15260.364} C_VEL
LIN {X 0,Y 319.564,Z 300.676,A -85,B 0,C 180,E1 -15264.456,E2 -15264.456} C_VEL
LIN {X 0,Y 319.504,Z 300.683,A -85,B 0,C 180,E1 -15268.134,E2 -15268.134} C_VEL
LIN {X 0,Y 319.576,Z 300.675,A -85,B 0,C 180,E1 -15271.595,E2 -15271.595} C_VEL
LIN {X 0,Y 319.555,Z 300.681,A -85,B 0,C 180,E1 -15275.299,E2 -15275.299} C_VEL
LIN {X 0,Y 319.545,Z 300.678,A -85,B 0,C 180,E1 -15278.043,E2 -15278.043} C_VEL
LIN {X 0,Y 319.593,Z 300.672,A -85,B 0,C 180,E1 -15282.069,E2 -15282.069} C_VEL
LIN {X 0,Y 319.709,Z 300.658,A -85,B 0,C 180,E1 -15286.006,E2 -15286.006} C_VEL
LIN {X 0,Y 319.714,Z 300.658,A -85,B 0,C 180,E1 -15289.871,E2 -15289.871} C_VEL
LIN {X 0,Y 319.916,Z 300.634,A -85,B 0,C 180,E1 -15293.693,E2 -15293.693} C_VEL
LIN {X 0,Y 319.96,Z 300.632,A -85,B 0,C 180,E1 -15297.482,E2 -15297.482} C_VEL
LIN {X 0,Y 320.072,Z 300.613,A -85,B 0,C 180,E1 -15299.999,E2 -15299.999} C_VEL
LIN {X 0,Y 319.96,Z 300.626,A -85,B 0,C 180,E1 -15302.517,E2 -15302.517} C_VEL
LIN {X 0,Y 319.877,Z 300.636,A -85,B 0,C 180,E1 -15306.71,E2 -15306.71} C_VEL
LIN {X 0,Y 319.73,Z 300.656,A -85,B 0,C 180,E1 -15310.127,E2 -15310.127} C_VEL
LIN {X 0,Y 319.708,Z 300.66,A -85,B 0,C 180,E1 -15313.993,E2 -15313.993} C_VEL
LIN {X 0,Y 319.578,Z 300.677,A -85,B 0,C 180,E1 -15317.931,E2 -15317.931} C_VEL
LIN {X 0,Y 319.544,Z 300.682,A -85,B 0,C 180,E1 -15321.955,E2 -15321.955} C_VEL
LIN {X 0,Y 319.615,Z 300.672,A -85,B 0,C 180,E1 -15326.089,E2 -15326.089} C_VEL
LIN {X 0,Y 319.57,Z 300.674,A -85,B 0,C 180,E1 -15328.935,E2 -15328.935} C_VEL
LIN {X 0,Y 319.514,Z 300.687,A -85,B 0,C 180,E1 -15331.863,E2 -15331.863} C_VEL
LIN {X 0,Y 319.563,Z 300.678,A -85,B 0,C 180,E1 -15335.543,E2 -15335.543} C_VEL
LIN {X 0,Y 319.559,Z 300.682,A -85,B 0,C 180,E1 -15338.009,E2 -15338.009} C_VEL
LIN {X 0,Y 319.517,Z 300.683,A -85,B 0,C 180,E1 -15341.599,E2 -15341.599} C_VEL
LIN {X 0,Y 319.547,Z 300.678,A -85,B 0,C 180,E1 -15345.271,E2 -15345.271} C_VEL
LIN {X 0,Y 319.568,Z 300.676,A -85,B 0,C 180,E1 -15348.72,E2 -15348.72} C_VEL
LIN {X 0,Y 319.589,Z 300.676,A -85,B 0,C 180,E1 -15352.34,E2 -15352.34} C_VEL
LIN {X 0,Y 319.552,Z 300.677,A -85,B 0,C 180,E1 -15355.124,E2 -15355.124} C_VEL
LIN {X 0,Y 319.559,Z 300.676,A -85,B 0,C 180,E1 -15359.06,E2 -15359.06} C_VEL
LIN {X 0,Y 319.6,Z 300.675,A -85,B 0,C 180,E1 -15362.498,E2 -15362.498} C_VEL
LIN {X 0,Y 319.6,Z 300.671,A -85,B 0,C 180,E1 -15365.304,E2 -15365.304} C_VEL
LIN {X 0,Y 319.593,Z 300.675,A -85,B 0,C 180,E1 -15368.048,E2 -15368.048} C_VEL
LIN {X 0,Y 319.686,Z 300.661,A -85,B 0,C 180,E1 -15370.962,E2 -15370.962} C_VEL
LIN {X 0,Y 319.728,Z 300.655,A -85,B 0,C 180,E1 -15375.275,E2 -15375.275} C_VEL
LIN {X 0,Y 319.756,Z 300.652,A -85,B 0,C 180,E1 -15379.872,E2 -15379.872} C_VEL
LIN {X 0,Y 319.931,Z 300.634,A -85,B 0,C 180,E1 -15382.425,E2 -15382.425} C_VEL
LIN {X 0,Y 319.744,Z 300.655,A -85,B 0,C 180,E1 -15384.955,E2 -15384.955} C_VEL
LIN {X 0,Y 319.988,Z 300.622,A -85,B 0,C 180,E1 -15387.481,E2 -15387.481} C_VEL
LIN {X 0,Y 320.148,Z 300.603,A -85,B 0,C 180,E1 -15389.998,E2 -15389.998} C_VEL
LIN {X 0,Y 319.988,Z 300.627,A -85,B 0,C 180,E1 -15392.515,E2 -15392.515} C_VEL
LIN {X 0,Y 319.946,Z 300.63,A -85,B 0,C 180,E1 -15396.303,E2 -15396.303} C_VEL
LIN {X 0,Y 319.837,Z 300.646,A -85,B 0,C 180,E1 -15398.845,E2 -15398.845} C_VEL
LIN {X 0,Y 319.678,Z 300.666,A -85,B 0,C 180,E1 -15402.697,E2 -15402.697} C_VEL
LIN {X 0,Y 319.691,Z 300.661,A -85,B 0,C 180,E1 -15405.292,E2 -15405.292} C_VEL
LIN {X 0,Y 319.68,Z 300.664,A -85,B 0,C 180,E1 -15409.251,E2 -15409.251} C_VEL
LIN {X 0,Y 319.562,Z 300.678,A -85,B 0,C 180,E1 -15413.315,E2 -15413.315} C_VEL
LIN {X 0,Y 319.621,Z 300.668,A -85,B 0,C 180,E1 -15416.084,E2 -15416.084} C_VEL
LIN {X 0,Y 319.574,Z 300.679,A -85,B 0,C 180,E1 -15418.93,E2 -15418.93} C_VEL
LIN {X 0,Y 319.514,Z 300.682,A -85,B 0,C 180,E1 -15421.858,E2 -15421.858} C_VEL
LIN {X 0,Y 319.559,Z 300.678,A -85,B 0,C 180,E1 -15425.539,E2 -15425.539} C_VEL
LIN {X 0,Y 319.614,Z 300.672,A -85,B 0,C 180,E1 -15428.371,E2 -15428.371} C_VEL
LIN {X 0,Y 328.347,Z 326.718,A -85,B 0,C 180,E1 -15429.618,E2 -15429.618} C_VEL
LIN {X 0,Y 325.998,Z 408.673,A -85,B 0,C 180,E1 -15431.774,E2 -15431.774} C_VEL
LIN {X 0,Y 325.521,Z 421.172,A -85,B 0,C 180,E1 -15432.333,E2 -15432.333} C_VEL
LIN {X 0,Y 324.818,Z 433.651,A -85,B 0,C 180,E1 -15433.122,E2 -15433.122} C_VEL
LIN {X 0,Y 323.927,Z 445.68,A -85,B 0,C 180,E1 -15434.143,E2 -15434.143} C_VEL
LIN {X 0,Y 322.895,Z 457.429,A -85,B 0,C 180,E1 -15435.418,E2 -15435.418} C_VEL
LIN {X 0,Y 321.96,Z 467.448,A -85,B 0,C 180,E1 -15436.775,E2 -15436.775} C_VEL
LIN {X 0,Y 320.936,Z 477.58,A -85,B 0,C 180,E1 -15438.485,E2 -15438.485} C_VEL
LIN {X 0,Y 320.077,Z 485.878,A -85,B 0,C 180,E1 -15440.209,E2 -15440.209} C_VEL
LIN {X 0,Y 319.389,Z 492.761,A -85,B 0,C 180,E1 -15441.967,E2 -15441.967} C_VEL
LIN {X 0,Y 318.951,Z 497.64,A -85,B 0,C 180,E1 -15443.493,E2 -15443.493} C_VEL
LIN {X 0,Y 318.552,Z 501.648,A -85,B 0,C 180,E1 -15444.998,E2 -15444.998} C_VEL
LIN {X 0,Y 318.424,Z 503.819,A -85,B 0,C 180,E1 -15445.962,E2 -15445.962} C_VEL
LIN {X 0,Y 317.575,Z 505.809,A -85,B 0,C 180,E1 -15446.955,E2 -15446.955} C_VEL
LIN {X 0,Y 314.427,Z 508.514,A -85,B 0,C 180,E1 -15448.591,E2 -15448.591} C_VEL
LIN {X 0,Y 311.859,Z 510.161,A -85,B 0,C 180,E1 -15449.941,E2 -15449.941} C_VEL
LIN {X 0,Y 310.796,Z 511.096,A -85,B 0,C 180,E1 -15451.001,E2 -15451.001} C_VEL
LIN {X 0,Y 310.726,Z 511.311,A -85,B 0,C 180,E1 -15451.362,E2 -15451.362} C_VEL
LIN {X 0,Y 310.76,Z 512.039,A -85,B 0,C 180,E1 -15453.109,E2 -15453.109} C_VEL
LIN {X 0,Y 310.929,Z 512.045,A -85,B 0,C 180,E1 -15454.689,E2 -15454.689} C_VEL
LIN {X 0,Y 311.132,Z 511.538,A -85,B 0,C 180,E1 -15456.01,E2 -15456.01} C_VEL
LIN {X 0,Y 311.517,Z 510.356,A -85,B 0,C 180,E1 -15457.646,E2 -15457.646} C_VEL
LIN {X 0,Y 312.126,Z 508.052,A -85,B 0,C 180,E1 -15459.574,E2 -15459.574} C_VEL
LIN {X 0,Y 312.9,Z 504.409,A -85,B 0,C 180,E1 -15461.673,E2 -15461.673} C_VEL
LIN {X 0,Y 314.226,Z 498.564,A -85,B 0,C 180,E1 -15464.072,E2 -15464.072} C_VEL
LIN {X 0,Y 315.673,Z 491.915,A -85,B 0,C 180,E1 -15466.153,E2 -15466.153} C_VEL
LIN {X 0,Y 317.184,Z 484.435,A -85,B 0,C 180,E1 -15467.995,E2 -15467.995} C_VEL
LIN {X 0,Y 319,Z 475.006,A -85,B 0,C 180,E1 -15469.849,E2 -15469.849} C_VEL
LIN {X 0,Y 320.738,Z 465.539,A -85,B 0,C 180,E1 -15471.336,E2 -15471.336} C_VEL
LIN {X 0,Y 322.484,Z 453.865,A -85,B 0,C 180,E1 -15472.802,E2 -15472.802} C_VEL
LIN {X 0,Y 323.996,Z 442.663,A -85,B 0,C 180,E1 -15473.909,E2 -15473.909} C_VEL
LIN {X 0,Y 325.166,Z 431.531,A -85,B 0,C 180,E1 -15474.774,E2 -15474.774} C_VEL
LIN {X 0,Y 326.23,Z 418.401,A -85,B 0,C 180,E1 -15475.522,E2 -15475.522} C_VEL
LIN {X 0,Y 326.924,Z 406.043,A -85,B 0,C 180,E1 -15475.994,E2 -15475.994} C_VEL
LIN {X 0,Y 330.22,Z 335.381,A -85,B 0,C 180,E1 -15478,E2 -15478} C_VEL
LIN {X 0,Y 322.297,Z 318.447,A -85,B 0,C 180,E1 -15479.659,E2 -15479.659} C_VEL
LIN {X 0,Y 315.82,Z 307.332,A -85,B 0,C 180,E1 -15481.05,E2 -15481.05} C_VEL
LIN {X 0,Y 313.523,Z 303.592,A -85,B 0,C 180,E1 -15481.606,E2 -15481.606} C_VEL
LIN {X 0,Y 312.913,Z 301.508,A -85,B 0,C 180,E1 -15482.414,E2 -15482.414} C_VEL
LIN {X 0,Y 312.853,Z 301.514,A -85,B 0,C 180,E1 -15486.45,E2 -15486.45} C_VEL
LIN {X 0,Y 312.716,Z 301.533,A -85,B 0,C 180,E1 -15489.052,E2 -15489.052} C_VEL
LIN {X 0,Y 312.591,Z 301.544,A -85,B 0,C 180,E1 -15492.994,E2 -15492.994} C_VEL
LIN {X 0,Y 312.58,Z 301.545,A -85,B 0,C 180,E1 -15495.653,E2 -15495.653} C_VEL
LIN {X 0,Y 312.496,Z 301.554,A -85,B 0,C 180,E1 -15499.716,E2 -15499.716} C_VEL
LIN {X 0,Y 312.5,Z 301.556,A -85,B 0,C 180,E1 -15503.88,E2 -15503.88} C_VEL
LIN {X 0,Y 312.5,Z 301.555,A -85,B 0,C 180,E1 -15506.731,E2 -15506.731} C_VEL
LIN {X 0,Y 312.473,Z 301.56,A -85,B 0,C 180,E1 -15509.658,E2 -15509.658} C_VEL
LIN {X 0,Y 312.489,Z 301.557,A -85,B 0,C 180,E1 -15513.693,E2 -15513.693} C_VEL
LIN {X 0,Y 312.511,Z 301.552,A -85,B 0,C 180,E1 -15517.388,E2 -15517.388} C_VEL
LIN {X 0,Y 312.468,Z 301.562,A -85,B 0,C 180,E1 -15520.713,E2 -15520.713} C_VEL
LIN {X 0,Y 312.428,Z 301.565,A -85,B 0,C 180,E1 -15524.215,E2 -15524.215} C_VEL
LIN {X 0,Y 312.463,Z 301.565,A -85,B 0,C 180,E1 -15527.924,E2 -15527.924} C_VEL
LIN {X 0,Y 312.484,Z 301.56,A -85,B 0,C 180,E1 -15530.976,E2 -15530.976} C_VEL
LIN {X 0,Y 312.521,Z 301.673,A -85,B 0,C 180,E1 -15532.81,E2 -15532.81} C_VEL
LIN {X 0,Y 315.026,Z 309.763,A -85,B 0,C 180,E1 -15535.634,E2 -15535.634} C_VEL
LIN {X 0,Y 317.312,Z 317.993,A -85,B 0,C 180,E1 -15538.269,E2 -15538.269} C_VEL
LIN {X 0,Y 319.328,Z 327.571,A -85,B 0,C 180,E1 -15541.046,E2 -15541.046} C_VEL
LIN {X 0,Y 319.579,Z 328.981,A -85,B 0,C 180,E1 -15541.436,E2 -15541.436} C_VEL
LIN {X 0,Y 321.201,Z 333.452,A -85,B 0,C 180,E1 -15541.833,E2 -15541.833} C_VEL
LIN {X 0,Y 325.04,Z 352.059,A -85,B 0,C 180,E1 -15543.023,E2 -15543.023} C_VEL
LIN {X 0,Y 327.553,Z 368.703,A -85,B 0,C 180,E1 -15543.91,E2 -15543.91} C_VEL
LIN {X 0,Y 328.621,Z 380.053,A -85,B 0,C 180,E1 -15544.423,E2 -15544.423} C_VEL
LIN {X 0,Y 325.748,Z 441.641,A -85,B 0,C 180,E1 -15546.185,E2 -15546.185} C_VEL
LIN {X 0,Y 324.464,Z 455.385,A -85,B 0,C 180,E1 -15546.804,E2 -15546.804} C_VEL
LIN {X 0,Y 322.952,Z 467.978,A -85,B 0,C 180,E1 -15547.619,E2 -15547.619} C_VEL
LIN {X 0,Y 321.172,Z 480.17,A -85,B 0,C 180,E1 -15548.671,E2 -15548.671} C_VEL
LIN {X 0,Y 319.388,Z 491.264,A -85,B 0,C 180,E1 -15549.894,E2 -15549.894} C_VEL
LIN {X 0,Y 317.62,Z 501.375,A -85,B 0,C 180,E1 -15551.29,E2 -15551.29} C_VEL
LIN {X 0,Y 315.881,Z 510.616,A -85,B 0,C 180,E1 -15552.859,E2 -15552.859} C_VEL
LIN {X 0,Y 314.321,Z 519.701,A -85,B 0,C 180,E1 -15554.772,E2 -15554.772} C_VEL
LIN {X 0,Y 313.002,Z 527.078,A -85,B 0,C 180,E1 -15556.698,E2 -15556.698} C_VEL
LIN {X 0,Y 312.01,Z 532.122,A -85,B 0,C 180,E1 -15558.307,E2 -15558.307} C_VEL
LIN {X 0,Y 311.363,Z 537.038,A -85,B 0,C 180,E1 -15560.257,E2 -15560.257} C_VEL
LIN {X 0,Y 310.978,Z 540.822,A -85,B 0,C 180,E1 -15562.21,E2 -15562.21} C_VEL
LIN {X 0,Y 310.819,Z 543.633,A -85,B 0,C 180,E1 -15564.213,E2 -15564.213} C_VEL
LIN {X 0,Y 310.8,Z 545.344,A -85,B 0,C 180,E1 -15566.113,E2 -15566.113} C_VEL
LIN {X 0,Y 310.79,Z 546.019,A -85,B 0,C 180,E1 -15567.41,E2 -15567.41} C_VEL
LIN {X 0,Y 310.903,Z 546.238,A -85,B 0,C 180,E1 -15568.707,E2 -15568.707} C_VEL
LIN {X 0,Y 311.077,Z 546.04,A -85,B 0,C 180,E1 -15570.002,E2 -15570.002} C_VEL
LIN {X 0,Y 310.991,Z 545.411,A -85,B 0,C 180,E1 -15571.297,E2 -15571.297} C_VEL
LIN {X 0,Y 310.856,Z 544.341,A -85,B 0,C 180,E1 -15572.593,E2 -15572.593} C_VEL
LIN {X 0,Y 310.879,Z 542.795,A -85,B 0,C 180,E1 -15573.89,E2 -15573.89} C_VEL
LIN {X 0,Y 310.934,Z 539.317,A -85,B 0,C 180,E1 -15575.993,E2 -15575.993} C_VEL
LIN {X 0,Y 311.021,Z 535.287,A -85,B 0,C 180,E1 -15577.793,E2 -15577.793} C_VEL
LIN {X 0,Y 311.387,Z 528.655,A -85,B 0,C 180,E1 -15580.075,E2 -15580.075} C_VEL
LIN {X 0,Y 311.992,Z 521.32,A -85,B 0,C 180,E1 -15582.028,E2 -15582.028} C_VEL
LIN {X 0,Y 312.905,Z 512.168,A -85,B 0,C 180,E1 -15583.973,E2 -15583.973} C_VEL
LIN {X 0,Y 313.793,Z 502.72,A -85,B 0,C 180,E1 -15585.591,E2 -15585.591} C_VEL
LIN {X 0,Y 314.944,Z 492.239,A -85,B 0,C 180,E1 -15587.031,E2 -15587.031} C_VEL
LIN {X 0,Y 316.072,Z 480.662,A -85,B 0,C 180,E1 -15588.305,E2 -15588.305} C_VEL
LIN {X 0,Y 317.144,Z 468.599,A -85,B 0,C 180,E1 -15589.331,E2 -15589.331} C_VEL
LIN {X 0,Y 318.208,Z 454.831,A -85,B 0,C 180,E1 -15590.188,E2 -15590.188} C_VEL
LIN {X 0,Y 318.924,Z 441.838,A -85,B 0,C 180,E1 -15590.73,E2 -15590.73} C_VEL
LIN {X 0,Y 320.579,Z 376.377,A -85,B 0,C 180,E1 -15592.498,E2 -15592.498} C_VEL
LIN {X 0,Y 315.554,Z 334.57,A -85,B 0,C 180,E1 -15594.005,E2 -15594.005} C_VEL
LIN {X 0,Y 316.832,Z 323.935,A -85,B 0,C 180,E1 -15596.636,E2 -15596.636} C_VEL
LIN {X 0,Y 315.659,Z 316.562,A -85,B 0,C 180,E1 -15598.599,E2 -15598.599} C_VEL
LIN {X 0,Y 312.624,Z 302.04,A -85,B 0,C 180,E1 -15602.651,E2 -15602.651} C_VEL
LIN {X 0,Y 312.556,Z 301.554,A -85,B 0,C 180,E1 -15602.83,E2 -15602.83} C_VEL
LIN {X 0,Y 312.529,Z 301.552,A -85,B 0,C 180,E1 -15605.947,E2 -15605.947} C_VEL
LIN {X 0,Y 312.45,Z 301.562,A -85,B 0,C 180,E1 -15610.113,E2 -15610.113} C_VEL
LIN {X 0,Y 312.448,Z 301.562,A -85,B 0,C 180,E1 -15613.962,E2 -15613.962} C_VEL
LIN {X 0,Y 312.426,Z 301.564,A -85,B 0,C 180,E1 -15617.927,E2 -15617.927} C_VEL
LIN {X 0,Y 312.463,Z 301.56,A -85,B 0,C 180,E1 -15621.923,E2 -15621.923} C_VEL
LIN {X 0,Y 312.516,Z 301.553,A -85,B 0,C 180,E1 -15624.218,E2 -15624.218} C_VEL
LIN {X 0,Y 312.486,Z 301.56,A -85,B 0,C 180,E1 -15627.331,E2 -15627.331} C_VEL
LIN {X 0,Y 312.507,Z 301.558,A -85,B 0,C 180,E1 -15631.285,E2 -15631.285} C_VEL
LIN {X 0,Y 312.531,Z 301.553,A -85,B 0,C 180,E1 -15634.706,E2 -15634.706} C_VEL
LIN {X 0,Y 312.5,Z 301.558,A -85,B 0,C 180,E1 -15638.909,E2 -15638.909} C_VEL
LIN {X 0,Y 312.547,Z 301.551,A -85,B 0,C 180,E1 -15641.65,E2 -15641.65} C_VEL
LIN {X 0,Y 312.664,Z 301.537,A -85,B 0,C 180,E1 -15645.684,E2 -15645.684} C_VEL
LIN {X 0,Y 312.664,Z 301.538,A -85,B 0,C 180,E1 -15649.64,E2 -15649.64} C_VEL
LIN {X 0,Y 312.822,Z 301.515,A -85,B 0,C 180,E1 -15652.252,E2 -15652.252} C_VEL
LIN {X 0,Y 312.874,Z 301.513,A -85,B 0,C 180,E1 -15653.551,E2 -15653.551} C_VEL
LIN {X 0,Y 312.907,Z 301.511,A -85,B 0,C 180,E1 -15657.425,E2 -15657.425} C_VEL
LIN {X 0,Y 313.029,Z 301.491,A -85,B 0,C 180,E1 -15659.999,E2 -15659.999} C_VEL
LIN {X 0,Y 312.907,Z 301.504,A -85,B 0,C 180,E1 -15662.574,E2 -15662.574} C_VEL
LIN {X 0,Y 312.839,Z 301.512,A -85,B 0,C 180,E1 -15666.694,E2 -15666.694} C_VEL
LIN {X 0,Y 312.737,Z 301.527,A -85,B 0,C 180,E1 -15669.05,E2 -15669.05} C_VEL
LIN {X 0,Y 312.61,Z 301.542,A -85,B 0,C 180,E1 -15672.991,E2 -15672.991} C_VEL
LIN {X 0,Y 312.598,Z 301.549,A -85,B 0,C 180,E1 -15675.651,E2 -15675.651} C_VEL
LIN {X 0,Y 312.514,Z 301.559,A -85,B 0,C 180,E1 -15679.713,E2 -15679.713} C_VEL
LIN {X 0,Y 312.517,Z 301.558,A -85,B 0,C 180,E1 -15683.877,E2 -15683.877} C_VEL
LIN {X 0,Y 312.535,Z 301.551,A -85,B 0,C 180,E1 -15686.726,E2 -15686.726} C_VEL
LIN {X 0,Y 312.527,Z 301.556,A -85,B 0,C 180,E1 -15689.651,E2 -15689.651} C_VEL
LIN {X 0,Y 312.504,Z 301.559,A -85,B 0,C 180,E1 -15693.689,E2 -15693.689} C_VEL
LIN {X 0,Y 312.511,Z 301.555,A -85,B 0,C 180,E1 -15697.386,E2 -15697.386} C_VEL
LIN {X 0,Y 312.48,Z 301.558,A -85,B 0,C 180,E1 -15700.71,E2 -15700.71} C_VEL
LIN {X 0,Y 312.468,Z 301.563,A -85,B 0,C 180,E1 -15704.206,E2 -15704.206} C_VEL
LIN {X 0,Y 312.537,Z 301.555,A -85,B 0,C 180,E1 -15707.907,E2 -15707.907} C_VEL
LIN {X 0,Y 312.548,Z 301.553,A -85,B 0,C 180,E1 -15711.906,E2 -15711.906} C_VEL
LIN {X 0,Y 312.499,Z 301.557,A -85,B 0,C 180,E1 -15715.79,E2 -15715.79} C_VEL
LIN {X 0,Y 312.513,Z 301.554,A -85,B 0,C 180,E1 -15718.854,E2 -15718.854} C_VEL
LIN {X 0,Y 312.565,Z 301.549,A -85,B 0,C 180,E1 -15721.825,E2 -15721.825} C_VEL
LIN {X 0,Y 312.581,Z 301.547,A -85,B 0,C 180,E1 -15724.711,E2 -15724.711} C_VEL
LIN {X 0,Y 312.584,Z 301.545,A -85,B 0,C 180,E1 -15727.529,E2 -15727.529} C_VEL
LIN {X 0,Y 312.636,Z 301.539,A -85,B 0,C 180,E1 -15731.656,E2 -15731.656} C_VEL
LIN {X 0,Y 312.691,Z 301.532,A -85,B 0,C 180,E1 -15735.685,E2 -15735.685} C_VEL
LIN {X 0,Y 312.7,Z 301.53,A -85,B 0,C 180,E1 -15739.641,E2 -15739.641} C_VEL
LIN {X 0,Y 312.87,Z 301.512,A -85,B 0,C 180,E1 -15742.253,E2 -15742.253} C_VEL
LIN {X 0,Y 312.715,Z 301.532,A -85,B 0,C 180,E1 -15744.841,E2 -15744.841} C_VEL
LIN {X 0,Y 312.988,Z 301.5,A -85,B 0,C 180,E1 -15748.711,E2 -15748.711} C_VEL
LIN {X 0,Y 312.988,Z 301.495,A -85,B 0,C 180,E1 -15751.284,E2 -15751.284} C_VEL
LIN {X 0,Y 312.714,Z 301.53,A -85,B 0,C 180,E1 -15755.155,E2 -15755.155} C_VEL
LIN {X 0,Y 312.867,Z 301.51,A -85,B 0,C 180,E1 -15757.743,E2 -15757.743} C_VEL
LIN {X 0,Y 312.665,Z 301.535,A -85,B 0,C 180,E1 -15761.668,E2 -15761.668} C_VEL
LIN {X 0,Y 312.692,Z 301.537,A -85,B 0,C 180,E1 -15764.884,E2 -15764.884} C_VEL
LIN {X 0,Y 312.635,Z 301.541,A -85,B 0,C 180,E1 -15769.241,E2 -15769.241} C_VEL
LIN {X 0,Y 312.536,Z 301.555,A -85,B 0,C 180,E1 -15772.787,E2 -15772.787} C_VEL
